// TwinCAT 3 PLC project Untitled1
// ProgramVersion: 3.1.4026.24
// libraries:
//   Tc2_MC2, * (Beckhoff Automation GmbH)
//   Tc2_Standard, * (Beckhoff Automation GmbH)
//   Tc2_System, * (Beckhoff Automation GmbH)
// project tree:
//   DUTs/ ST_ServiceCtrlBase.TcDUT, ST_ServiceStatusBase.TcDUT
//   GVLs/ GVL_Remote.TcGVL
//   / PlcTask.TcTTO
//   POUs/00_BaseUnit/ FB_AxisControl.TcPOU, FB_BaseUnit.TcPOU, T_ResourceOwnerId.TcDUT
//   POUs/10_Module/11_GC/DUTs/ E_GCResourceOwnerId.TcDUT, ST_GC_Admin.TcDUT, ST_GC_ServiceCtrl.TcDUT, ST_GC_ServiceStatus.TcDUT
//   POUs/10_Module/11_GC/DUTs/SpinAxisJogService/ E_GCSpinAxisJogErrorCode.TcDUT, ST_GCSpinAxisJogCtrl.TcDUT, ST_GCSpinAxisJogParam.TcDUT, ST_GCSpinAxisJogStatus.TcDUT
//   POUs/10_Module/11_GC/DUTs/SpinAxisMoveAbsService/ E_GCSpinAxisMoveAbsErrorCode.TcDUT, ST_GCSpinAxisMoveAbsCtrl.TcDUT, ST_GCSpinAxisMoveAbsParam.TcDUT (not stored), ST_GCSpinAxisMoveAbsStatus.TcDUT
//   POUs/10_Module/11_GC/DUTs/SpinAxisMoveVelService/ E_GCSpinAxisMoveVelErrorCode.TcDUT, ST_GCSpinAxisMoveVelCtrl.TcDUT (not stored), ST_GCSpinAxisMoveVelParam.TcDUT, ST_GCSpinAxisMoveVelStatus.TcDUT
//   POUs/10_Module/11_GC/ FB_GC.TcPOU
//   POUs/10_Module/11_GC/Services/ FB_GCSpinAxisJogServices.TcPOU, FB_GCSpinAxisMoveAbsServices.TcPOU, FB_GCSpinAxisMoveVelServices.TcPOU
//   POUs/20_Machine/DUTs/ ST_Machine_Admin.TcDUT, ST_Machine_Ctrl.TcDUT, ST_Machine_ServiceCtrl.TcDUT, ST_Machine_ServiceStatus.TcDUT, ST_Machine_Status.TcDUT
//   POUs/20_Machine/ FB_Machine.TcPOU
//   POUs/ MAIN.TcPOU
//   POUs/PackML_Base/DUTs/ E_PackMLCommand.TcDUT (not stored), E_PackMLHookResult.TcDUT (not stored), E_PackMLMode.TcDUT (not stored), E_PackMLState.TcDUT (not stored), ST_PML_Base_In.TcDUT, ST_PML_Base_Out.TcDUT, T_PackMLMode.TcDUT (not stored)
//   POUs/PackML_Base/ FB_PackMLBase.TcPOU, FB_PackMLModeSet.TcPOU, I_ModuleServiceProperty.TcIO
//   POUs/PackML_Base/Utilities/ F_PackMLCommandToString.TcPOU, F_PackMLModeToString.TcPOU, F_PackMLStateToString.TcPOU (not stored)
// real-time tasks:
//   TASK PlcTask: cycle T#10ms, priority 20, ADS port 350
// motion (NC):
//   TASK NC-Task 1 SAF: cycle T#2ms, priority 4, ADS port 501
//   TASK NC-Task 1 SVB: cycle T#10ms, priority 8, ADS port 511
//   AXIS Axis 1 (id 1)
//     OtherSettings: AllowMotionCmdToSlave=true
//     encoder EncType=1
//     drive DrvType=5
//       Analog: TorqueSetpointScale=10, ScaleFactorActTorque=0.1
//       TimeComp: TaskDelayCycles=1
//     controller CtrType=1
//       CtrPara: PriorControlFactor=1
//         Observer: BandWidth=20
// variable links:
//   Untitled1/Untitled1 Instance <-> NC-Task 1 SAF/Axes/Axis 1
//     PlcTask Inputs/MAIN.Machine._GCSpinAxis.NcToPlc <-> Outputs/ToPlc
//     PlcTask Outputs/MAIN.Machine._GCSpinAxis.PlcToNc <-> Inputs/FromPlc

CONFIGURATION Untitled1
    RESOURCE PLC ON TwinCAT3
        TASK PlcTask(INTERVAL := T#10ms, PRIORITY := 20);
        PROGRAM MAIN WITH PlcTask : MAIN;
    END_RESOURCE
END_CONFIGURATION

// ---- DUTs/ST_ServiceCtrlBase.TcDUT
TYPE ST_ServiceCtrlBase :
STRUCT
	Start : BOOL;
	Reset : BOOL;
	Stop : BOOL;
	Abort : BOOL;
END_STRUCT
END_TYPE

// ---- DUTs/ST_ServiceStatusBase.TcDUT
TYPE ST_ServiceStatusBase :
STRUCT
	Busy : BOOL;
	Done : BOOL;
	Error : BOOL;
	Aborted : BOOL;
	ErrorId : UDINT;
	State : E_PackMLState;
END_STRUCT
END_TYPE

// ---- POUs/00_BaseUnit/T_ResourceOwnerId.TcDUT
// Zero is reserved to represent an unowned resource.
TYPE T_ResourceOwnerId : UDINT;
END_TYPE

// ---- POUs/10_Module/11_GC/DUTs/E_GCResourceOwnerId.TcDUT
{attribute 'qualified_only'}
{attribute 'to_string'}
TYPE E_GCResourceOwnerId :
(
	// Each value identifies one Service instance within the GC Module.
	None := 0,
	SpinAxisJog := 1,
	SpinAxisMoveAbs := 2,
	SpinAxisMoveVel := 3
) UDINT;
END_TYPE

// ---- POUs/10_Module/11_GC/DUTs/SpinAxisJogService/E_GCSpinAxisJogErrorCode.TcDUT
{attribute 'qualified_only'}
{attribute 'to_string'}
TYPE E_GCSpinAxisJogErrorCode :
(
	None := 0,
	Axis_Not_Servo_On_During_Starting,
	Axis_Is_Busy_During_Starting,
	Invalid_Param,
	Jog_Error_During_Execute,
	// The BaseUnit was already owned by another Service.
	Resource_Acquire_Failed_During_Starting
)UDINT;
END_TYPE

// ---- POUs/10_Module/11_GC/DUTs/SpinAxisJogService/ST_GCSpinAxisJogCtrl.TcDUT
TYPE ST_GCSpinAxisJogCtrl EXTENDS ST_ServiceCtrlBase:
STRUCT
	Param : ST_GCSpinAxisJogParam;
END_STRUCT
END_TYPE

// ---- POUs/10_Module/11_GC/DUTs/SpinAxisJogService/ST_GCSpinAxisJogParam.TcDUT
TYPE ST_GCSpinAxisJogParam :
STRUCT
	JogForward : BOOL;
	JogBackwards : BOOL;
	Mode : E_JogMode;
	Position : LREAL;
	Velocity : LREAL;
	Acceleration : LREAL;
	Deceleration : LREAL;
END_STRUCT
END_TYPE

// ---- POUs/10_Module/11_GC/DUTs/SpinAxisJogService/ST_GCSpinAxisJogStatus.TcDUT
TYPE ST_GCSpinAxisJogStatus EXTENDS ST_ServiceStatusBase :
STRUCT
END_STRUCT
END_TYPE

// ---- POUs/10_Module/11_GC/DUTs/SpinAxisMoveAbsService/E_GCSpinAxisMoveAbsErrorCode.TcDUT
{attribute 'qualified_only'}
{attribute 'to_string'}
TYPE E_GCSpinAxisMoveAbsErrorCode :
(
	None := 0,
	Axis_Not_Servo_On_During_Starting,
	Axis_Is_Busy_During_Starting,
	Invalid_Param,
	MoveAbs_Error_During_Execute,
	Error_While_Stop_Axis,
	// The BaseUnit was already owned by another Service.
	Resource_Acquire_Failed_During_Starting
)UDINT;
END_TYPE

// ---- POUs/10_Module/11_GC/DUTs/SpinAxisMoveAbsService/ST_GCSpinAxisMoveAbsCtrl.TcDUT
TYPE ST_GCSpinAxisMoveAbsCtrl EXTENDS ST_ServiceCtrlBase:
STRUCT
	Param : ST_GCSpinAxisMoveAbsParam;
END_STRUCT
END_TYPE

// ---- POUs/10_Module/11_GC/DUTs/SpinAxisMoveAbsService/ST_GCSpinAxisMoveAbsStatus.TcDUT
TYPE ST_GCSpinAxisMoveAbsStatus EXTENDS ST_ServiceStatusBase :
STRUCT
END_STRUCT
END_TYPE

// ---- POUs/10_Module/11_GC/DUTs/SpinAxisMoveVelService/E_GCSpinAxisMoveVelErrorCode.TcDUT
{attribute 'qualified_only'}
{attribute 'to_string'}
TYPE E_GCSpinAxisMoveVelErrorCode :
(
	None := 0,
	Axis_Not_Servo_On_During_Starting,
	Axis_Is_Busy_During_Starting,
	Invalid_Param,
	MoveVel_Error_During_Execute,
	Error_While_Stop_Axis,
	// The BaseUnit was already owned by another Service.
	Resource_Acquire_Failed_During_Starting
)UDINT;
END_TYPE

// ---- POUs/10_Module/11_GC/DUTs/SpinAxisMoveVelService/ST_GCSpinAxisMoveVelParam.TcDUT
TYPE ST_GCSpinAxisMoveVelParam :
STRUCT
	IsPositiveDirection	: BOOL;
	Velocity : LREAL;
	Acceleration : LREAL;
	Deceleration : LREAL;
END_STRUCT
END_TYPE

// ---- POUs/10_Module/11_GC/DUTs/SpinAxisMoveVelService/ST_GCSpinAxisMoveVelStatus.TcDUT
TYPE ST_GCSpinAxisMoveVelStatus EXTENDS ST_ServiceStatusBase :
STRUCT
	ActVel	: LREAL;
END_STRUCT
END_TYPE

// ---- POUs/10_Module/11_GC/DUTs/ST_GC_Admin.TcDUT
TYPE ST_GC_Admin :
STRUCT
	bLocalControl : BOOL;
END_STRUCT
END_TYPE

// ---- POUs/10_Module/11_GC/DUTs/ST_GC_ServiceCtrl.TcDUT
TYPE ST_GC_ServiceCtrl :
STRUCT
	SpinAxisJog : ST_GCSpinAxisJogCtrl;
	SpinAxisMoveAbs : ST_GCSpinAxisMoveAbsCtrl;
	SpinAxisMoveVel	: ST_GCSpinAxisMoveVelCtrl;
END_STRUCT
END_TYPE

// ---- POUs/10_Module/11_GC/DUTs/ST_GC_ServiceStatus.TcDUT
TYPE ST_GC_ServiceStatus :
STRUCT
	SpinAxisJog : ST_GCSpinAxisJogStatus;
	SpinAxisMoveAbs : ST_GCSpinAxisMoveAbsStatus;
	SpinAxisMoveVel : ST_GCSpinAxisMoveVelStatus;
END_STRUCT
END_TYPE

// ---- POUs/20_Machine/DUTs/ST_Machine_Admin.TcDUT
TYPE ST_Machine_Admin :
STRUCT
	GC_Admin : ST_GC_Admin;
END_STRUCT
END_TYPE

// ---- POUs/20_Machine/DUTs/ST_Machine_Ctrl.TcDUT
TYPE ST_Machine_Ctrl:
STRUCT
	Machine_Ctrl :ST_PML_Base_In;
	GC_Ctrl : ST_PML_Base_In;
END_STRUCT
END_TYPE

// ---- POUs/20_Machine/DUTs/ST_Machine_ServiceCtrl.TcDUT
TYPE ST_Machine_ServiceCtrl :
STRUCT
	GC : ST_GC_ServiceCtrl;
END_STRUCT
END_TYPE

// ---- POUs/20_Machine/DUTs/ST_Machine_ServiceStatus.TcDUT
TYPE ST_Machine_ServiceStatus :
STRUCT
	GC : ST_GC_ServiceStatus;
END_STRUCT
END_TYPE

// ---- POUs/20_Machine/DUTs/ST_Machine_Status.TcDUT
TYPE ST_Machine_Status:
STRUCT
	Machine_Status : ST_PML_Base_Out;
	GC_Status : ST_PML_Base_Out;
END_STRUCT
END_TYPE

// ---- POUs/PackML_Base/DUTs/ST_PML_Base_In.TcDUT
TYPE ST_PML_Base_In :
STRUCT
	eCommand				: E_PackMLCommand := E_PackMLCommand.None;
	bCommandChangeRequest	: BOOL;
	eMode					: T_PackMLMode := GVL_PackMLMode.Unknown;
	bModeChangeRequest	: BOOL;
END_STRUCT
END_TYPE

// ---- POUs/PackML_Base/DUTs/ST_PML_Base_Out.TcDUT
TYPE ST_PML_Base_Out :
STRUCT
	eStateCurrent		: E_PackMLState := E_PackMLState.Undefined;
	eStatePrevious		: E_PackMLState := E_PackMLState.Undefined;
	eModeCurrent		: T_PackMLMode := E_PackMLMode.Unknown;
	eModePrevious		: T_PackMLMode := E_PackMLMode.Unknown;

	bCommandAccepted	: BOOL;
	bCommandRejected	: BOOL;

	bModeChanged		: BOOL;
	bModeChangeRejected	: BOOL;
END_STRUCT
END_TYPE

// ---- GVLs/GVL_Remote.TcGVL
{attribute 'qualified_only'}
VAR_GLOBAL
	Ctrl : ST_Machine_Ctrl;
	Status : ST_Machine_Status;
	ServiceCtrl : ST_Machine_ServiceCtrl;
	ServiceStatus : ST_Machine_ServiceStatus;
	Admin : ST_Machine_Admin;
END_VAR

// ---- POUs/PackML_Base/I_ModuleServiceProperty.TcIO
INTERFACE I_ModuleServiceProperty

PROPERTY ModuleMode : T_PackMLMode
GET
END_GET
SET
END_SET
END_PROPERTY

END_INTERFACE

// ---- POUs/MAIN.TcPOU
PROGRAM MAIN
VAR
	Machine : FB_Machine;
END_VAR

Machine(
	Ctrl:= GVL_Remote.Ctrl, 
	Status:= GVL_Remote.Status, 
	ServiceCtrl:= GVL_Remote.ServiceCtrl,
	ServiceStatus:= GVL_Remote.ServiceStatus,
	Admin:= GVL_Remote.Admin);

END_PROGRAM

// ---- POUs/20_Machine/FB_Machine.TcPOU
FUNCTION_BLOCK FB_Machine EXTENDS FB_PackMLModeSet
VAR_INPUT
	Ctrl : REFERENCE TO ST_Machine_Ctrl;
	Status : REFERENCE TO ST_Machine_Status;
	ServiceCtrl : REFERENCE TO ST_Machine_ServiceCtrl;
	ServiceStatus : REFERENCE TO ST_Machine_ServiceStatus;
	Admin : REFERENCE TO ST_Machine_Admin;
END_VAR
VAR_OUTPUT
END_VAR
VAR
	// 有需要特殊操作的需求，所以建立一個ST_Machine_Ctrl變數，讓程式內部可以過一手處理
	_Ctrl : ST_Machine_Ctrl;
	
	// Module
	_GC_Module : FB_GC;
	
	// Component
	_GCSpinAxis : AXIS_REF;
	_GCSpinAxis_BaseUnit : FB_AxisControl;
END_VAR

stIn := Ctrl.Machine_Ctrl;
Status.Machine_Status := stOut;

// Select control source
IF Admin.GC_Admin.bLocalControl THEN
	_Ctrl.GC_Ctrl := Ctrl.GC_Ctrl;
ELSE
	_Ctrl.GC_Ctrl := Ctrl.Machine_Ctrl;
END_IF

A00_BaseUnit();
A01_Module();
A02_CompoundService();

SUPER^();

ACTION A00_BaseUnit:
_GCSpinAxis_BaseUnit(Axis:= _GCSpinAxis);
END_ACTION

ACTION A01_Module:
_GC_Module(
	stIn:= _Ctrl.GC_Ctrl,
	stOut=> Status.GC_Status,
	ServiceCtrl:= ServiceCtrl.GC,
	ServiceStatus:= ServiceStatus.GC,
	Admin:= Admin.GC_Admin,
	SpinAxis_BaseUnit:= _GCSpinAxis_BaseUnit);
END_ACTION

ACTION A02_CompoundService:

END_ACTION

METHOD PROTECTED H_OnAborted
VAR_INPUT
	bFirstScan	: BOOL;
END_VAR
END_METHOD

METHOD PROTECTED H_OnAborting : E_PackMLHookResult
VAR_INPUT
	bFirstScan	: BOOL;
END_VAR
// Default transient hooks complete immediately; override when work is required.
H_OnAborting := E_PackMLHookResult.Done;
END_METHOD

METHOD PROTECTED H_OnClearing : E_PackMLHookResult
VAR_INPUT
	bFirstScan	: BOOL;
END_VAR
H_OnClearing := E_PackMLHookResult.Busy;

// Wait cmd finished
IF Status.GC_Status.eStateCurrent <> E_PackMLState.Stopped THEN
	RETURN;
END_IF

H_OnClearing := E_PackMLHookResult.Done;
END_METHOD

METHOD PROTECTED H_OnComplete
VAR_INPUT
	bFirstScan	: BOOL;
END_VAR
// Default action hook intentionally empty. Override in derived FBs when needed.
END_METHOD

METHOD PROTECTED H_OnCompleting : E_PackMLHookResult
VAR_INPUT
	bFirstScan	: BOOL;
END_VAR
// Default transient hooks complete immediately; override when work is required.
H_OnCompleting := E_PackMLHookResult.Done;
END_METHOD

METHOD PROTECTED H_OnExecute : E_PackMLHookResult
VAR_INPUT
	bFirstScan	: BOOL;
END_VAR
// Execute is stable by default; derived FBs decide when the process is done.
H_OnExecute := E_PackMLHookResult.Busy;
END_METHOD

METHOD PROTECTED H_OnHeld
VAR_INPUT
	bFirstScan	: BOOL;
END_VAR
// Default action hook intentionally empty. Override in derived FBs when needed.
END_METHOD

METHOD PROTECTED H_OnHolding : E_PackMLHookResult
VAR_INPUT
	bFirstScan	: BOOL;
END_VAR
// Default transient hooks complete immediately; override when work is required.
H_OnHolding := E_PackMLHookResult.Done;
END_METHOD

METHOD PROTECTED H_OnIdle
VAR_INPUT
	bFirstScan	: BOOL;
END_VAR
END_METHOD

METHOD PROTECTED H_OnResetting : E_PackMLHookResult
VAR_INPUT
	bFirstScan	: BOOL;
END_VAR
H_OnResetting := E_PackMLHookResult.Busy;

// Wait cmd finished
IF Status.GC_Status.eStateCurrent <> E_PackMLState.Idle THEN
	RETURN;
END_IF

H_OnResetting := E_PackMLHookResult.Done;
END_METHOD

METHOD PROTECTED H_OnStarting : E_PackMLHookResult
VAR_INPUT
	bFirstScan	: BOOL;
END_VAR
H_OnStarting := E_PackMLHookResult.Busy;

// Wait cmd finished
IF Status.GC_Status.eStateCurrent <> E_PackMLState.Execute THEN
	RETURN;
END_IF

H_OnStarting := E_PackMLHookResult.Done;
END_METHOD

METHOD PROTECTED H_OnStopped
VAR_INPUT
	bFirstScan	: BOOL;
END_VAR
END_METHOD

METHOD PROTECTED H_OnStopping : E_PackMLHookResult
VAR_INPUT
	bFirstScan	: BOOL;
END_VAR
H_OnStopping := E_PackMLHookResult.Busy;

// Wait cmd finished
IF Status.GC_Status.eStateCurrent <> E_PackMLState.Stopped THEN
	RETURN;
END_IF

H_OnStopping := E_PackMLHookResult.Done;
END_METHOD

METHOD PROTECTED H_OnSuspended
VAR_INPUT
	bFirstScan	: BOOL;
END_VAR
// Default action hook intentionally empty. Override in derived FBs when needed.
END_METHOD

METHOD PROTECTED H_OnSuspending : E_PackMLHookResult
VAR_INPUT
	bFirstScan	: BOOL;
END_VAR
// Default transient hooks complete immediately; override when work is required.
H_OnSuspending := E_PackMLHookResult.Done;
END_METHOD

METHOD PROTECTED H_OnUndefined : E_PackMLHookResult
VAR_INPUT
	bFirstScan	: BOOL;
END_VAR
// The base FB leaves Undefined immediately unless a derived FB delays startup.
H_OnUndefined := E_PackMLHookResult.Done;
END_METHOD

METHOD PROTECTED H_OnUnholding : E_PackMLHookResult
VAR_INPUT
	bFirstScan	: BOOL;
END_VAR
// Default transient hooks complete immediately; override when work is required.
H_OnUnholding := E_PackMLHookResult.Done;
END_METHOD

METHOD PROTECTED H_OnUnsuspending : E_PackMLHookResult
VAR_INPUT
	bFirstScan	: BOOL;
END_VAR
// Default transient hooks complete immediately; override when work is required.
H_OnUnsuspending := E_PackMLHookResult.Done;
END_METHOD

END_FUNCTION_BLOCK

// ---- POUs/PackML_Base/FB_PackMLModeSet.TcPOU
FUNCTION_BLOCK FB_PackMLModeSet EXTENDS FB_PackMLBase
VAR_INPUT
END_VAR
VAR_OUTPUT
END_VAR
VAR
END_VAR

SUPER^();

METHOD PROTECTED H_IsCommandAllowedByMode : BOOL
VAR_INPUT
	eRequestedCommand	: E_PackMLCommand;
	eActiveMode	: T_PackMLMode;
END_VAR
CASE eActiveMode OF
	GVL_PackMLMode.Manual:
		// Supported commands in manual mode
		CASE eRequestedCommand OF
			E_PackMLCommand.Reset,
			E_PackMLCommand.Start,
			E_PackMLCommand.Stop,
			E_PackMLCommand.Abort,
			E_PackMLCommand.Clear:
				H_IsCommandAllowedByMode := TRUE;
			ELSE
				H_IsCommandAllowedByMode := FALSE;
		END_CASE
	
	GVL_PackMLMode.Production,
	GVL_PackMLMode.Unknown:
		// Support all commands in production mode
		H_IsCommandAllowedByMode := TRUE;
END_CASE
END_METHOD

METHOD PROTECTED H_IsModeSupported : BOOL
VAR_INPUT
	eRequestedMode	: T_PackMLMode;
END_VAR
CASE eRequestedMode OF
	GVL_PackMLMode.Manual,
	GVL_PackMLMode.Production:
		H_IsModeSupported := TRUE;

	ELSE
		H_IsModeSupported := FALSE;
END_CASE
END_METHOD

METHOD PROTECTED H_IsStateSupportedByMode : BOOL
VAR_INPUT
	eRequestedMode	: T_PackMLMode;
	eCurrentState	: E_PackMLState;
END_VAR
CASE eRequestedMode OF
	
	GVL_PackMLMode.Manual:
		// Support states in manual mode
		CASE eCurrentState OF
			E_PackMLState.Idle,
			E_PackMLState.Starting,
			E_PackMLState.Execute,
			E_PackMLState.Aborting,
			E_PackMLState.Aborted,
			E_PackMLState.Clearing,
			E_PackMLState.Stopped,
			E_PackMLState.Resetting:
			H_IsStateSupportedByMode := TRUE;
			
			ELSE
				H_IsStateSupportedByMode := FALSE;
		END_CASE
		
	
	GVL_PackMLMode.Production,
	GVL_PackMLMode.Unknown:
		// Support all state in production mode
		H_IsStateSupportedByMode := TRUE;
END_CASE
END_METHOD

END_FUNCTION_BLOCK

// ---- POUs/PackML_Base/FB_PackMLBase.TcPOU
FUNCTION_BLOCK FB_PackMLBase
VAR_INPUT
	stIn	: ST_PML_Base_In;
	
	bEnable				: BOOL := TRUE;
	bExternalFault		: BOOL;
END_VAR
VAR_OUTPUT
	stOut	: ST_PML_Base_Out;
	
	sStateErrorText		: STRING(255);
	sModeErrorText		: STRING(255);
	bTransitionActive	: BOOL;
END_VAR
VAR
	_eLastCommand			: E_PackMLCommand := E_PackMLCommand.None;
	_eCommandToProcess		: E_PackMLCommand := E_PackMLCommand.None;
	_eQueuedCommand			: E_PackMLCommand := E_PackMLCommand.None;
	_bQueuedCommandRequest	: BOOL;
	_bCommandConsumed		: BOOL;
	_bModeChangeConsumed	: BOOL;
	_bStateFirstScan		: BOOL := TRUE;
	_bStateFirstScanForHook	: BOOL;
	_eHookResult			: E_PackMLHookResult;
END_VAR

// Reset edge-style status before evaluating this PLC cycle.
_eCommandToProcess		:= E_PackMLCommand.None;

// Command and mode request feedback is latched for HMI/upper-layer handshakes
// until the corresponding request input returns to FALSE.
IF NOT stIn.bCommandChangeRequest THEN
	stOut.bCommandAccepted	:= FALSE;
	stOut.bCommandRejected	:= FALSE;
	sStateErrorText			:= '';
END_IF

IF NOT stIn.bModeChangeRequest THEN
	stOut.bModeChanged		:= FALSE;
	stOut.bModeChangeRejected	:= FALSE;
	sModeErrorText		:= '';
END_IF

// A disabled base FB holds the current state and suppresses transition activity.
IF NOT bEnable THEN
	bTransitionActive := FALSE;
	RETURN;
END_IF

// Mode change requests are edge/latch based, matching command request behavior.
// The caller must clear stIn.bModeChangeRequest before the same request can run again.
IF NOT stIn.bModeChangeRequest THEN
	_bModeChangeConsumed := FALSE;
END_IF

IF stIn.bModeChangeRequest AND NOT _bModeChangeConsumed THEN
	_bModeChangeConsumed := TRUE;

	IF NOT H_IsModeSupported(stIn.eMode) THEN
		M_RejectModeChange('Requested mode is not supported.');
	ELSIF stIn.eMode = stOut.eModeCurrent THEN
		M_RejectModeChange('Requested mode is already active.');
	ELSIF NOT M_IsModeChangeAllowedByState() THEN
		M_RejectModeChange('Mode change is only allowed from Aborted, Stopped, Idle, or Complete.');
	ELSIF NOT H_IsStateSupportedByMode(stIn.eMode, stOut.eStateCurrent) THEN
		M_RejectModeChange('Requested mode does not support the current PackML state.');
	ELSE
		M_ChangeMode(stIn.eMode);
	END_IF
END_IF

// Command requests are edge/latch based, matching mode-change request behavior.
// The caller must clear stIn.bCommandChangeRequest before another command can run.
IF NOT stIn.bCommandChangeRequest THEN
	_bCommandConsumed	:= FALSE;
	_eLastCommand		:= E_PackMLCommand.None;
END_IF

// External faults have priority over normal commands and force the abort path
// only while the machine is not already Aborting or Aborted.
IF bExternalFault AND M_IsAbortAllowedByState() THEN
	_eCommandToProcess := E_PackMLCommand.Abort;
ELSIF _bQueuedCommandRequest AND (_eQueuedCommand <> E_PackMLCommand.None) THEN
	_eCommandToProcess		:= _eQueuedCommand;
	_eQueuedCommand			:= E_PackMLCommand.None;
	_bQueuedCommandRequest	:= FALSE;
ELSIF stIn.bCommandChangeRequest AND (stIn.eCommand <> E_PackMLCommand.None) AND NOT _bCommandConsumed THEN
	_eCommandToProcess	:= stIn.eCommand;
	_eLastCommand		:= stIn.eCommand;
	_bCommandConsumed	:= TRUE;
END_IF

// Mode policy hooks run before PackML state guards so a forbidden command reports
// the mode reason instead of a state reason.
IF (_eCommandToProcess <> E_PackMLCommand.None) AND NOT H_IsCommandAllowedByMode(_eCommandToProcess, stOut.eModeCurrent) THEN
	M_RejectCommand(M_BuildCommandRejectedByModeText(_eCommandToProcess, stOut.eModeCurrent));
	_eCommandToProcess := E_PackMLCommand.None;
END_IF

// Dispatch the accepted command through private PackML state guards.
// Rejected commands never mutate the state and return a readable error text.
CASE _eCommandToProcess OF
	E_PackMLCommand.Clear:
		IF M_IsClearAllowedByState() THEN
			stOut.bCommandAccepted := TRUE;
			M_ChangeState(E_PackMLState.Clearing);
		ELSE
			M_RejectCommand('Clear command is only valid from Aborted.');
		END_IF

	E_PackMLCommand.Reset:
		IF M_IsResetAllowedByState() THEN
			stOut.bCommandAccepted := TRUE;
			M_ChangeState(E_PackMLState.Resetting);
		ELSE
			M_RejectCommand('Reset command is only valid from Stopped or Complete.');
		END_IF

	E_PackMLCommand.Start:
		IF M_IsStartAllowedByState() THEN
			stOut.bCommandAccepted := TRUE;
			M_ChangeState(E_PackMLState.Starting);
		ELSE
			M_RejectCommand('Start command is only valid from Idle.');
		END_IF

	E_PackMLCommand.Stop:
		IF M_IsStopAllowedByState() THEN
			stOut.bCommandAccepted := TRUE;
			M_ChangeState(E_PackMLState.Stopping);
		ELSE
			M_RejectCommand('Stop command is not valid from the current PackML state.');
		END_IF

	E_PackMLCommand.Hold:
		IF M_IsHoldAllowedByState() THEN
			stOut.bCommandAccepted := TRUE;
			M_ChangeState(E_PackMLState.Holding);
		ELSE
			M_RejectCommand('Hold command is only valid from Execute.');
		END_IF

	E_PackMLCommand.Unhold:
		IF M_IsUnholdAllowedByState() THEN
			stOut.bCommandAccepted := TRUE;
			M_ChangeState(E_PackMLState.Unholding);
		ELSE
			M_RejectCommand('Unhold command is only valid from Held.');
		END_IF

	E_PackMLCommand.Suspend:
		IF M_IsSuspendAllowedByState() THEN
			stOut.bCommandAccepted := TRUE;
			M_ChangeState(E_PackMLState.Suspending);
		ELSE
			M_RejectCommand('Suspend command is only valid from Execute.');
		END_IF

	E_PackMLCommand.Unsuspend:
		IF M_IsUnsuspendAllowedByState() THEN
			stOut.bCommandAccepted := TRUE;
			M_ChangeState(E_PackMLState.Unsuspending);
		ELSE
			M_RejectCommand('Unsuspend command is only valid from Suspended.');
		END_IF

	E_PackMLCommand.Abort:
		IF M_IsAbortAllowedByState() THEN
			stOut.bCommandAccepted := TRUE;
			M_ChangeState(E_PackMLState.Aborting);
		ELSE
			M_RejectCommand('Abort command is not valid while already Aborting or Aborted.');
		END_IF
END_CASE

// Run the current state's action hook, then advance transient states when their
// hook reports Done. Stable states remain active until a command moves them.
_bStateFirstScanForHook	:= _bStateFirstScan;
_bStateFirstScan		:= FALSE;

CASE stOut.eStateCurrent OF
	E_PackMLState.Undefined:
		_eHookResult := H_OnUndefined(_bStateFirstScanForHook);
		IF _eHookResult = E_PackMLHookResult.Done THEN
			M_ChangeState(E_PackMLState.Aborted);
		END_IF

	E_PackMLState.Clearing:
		_eHookResult := H_OnClearing(_bStateFirstScanForHook);
		IF _eHookResult = E_PackMLHookResult.Done THEN
			M_ChangeState(E_PackMLState.Stopped);
		END_IF

	E_PackMLState.Stopped:
		H_OnStopped(_bStateFirstScanForHook);

	E_PackMLState.Starting:
		_eHookResult := H_OnStarting(_bStateFirstScanForHook);
		IF _eHookResult = E_PackMLHookResult.Done THEN
			M_ChangeState(E_PackMLState.Execute);
		END_IF

	E_PackMLState.Idle:
		H_OnIdle(_bStateFirstScanForHook);

	E_PackMLState.Suspended:
		H_OnSuspended(_bStateFirstScanForHook);

	E_PackMLState.Execute:
		_eHookResult := H_OnExecute(_bStateFirstScanForHook);
		IF _eHookResult = E_PackMLHookResult.Done THEN
			M_ChangeState(E_PackMLState.Completing);
		END_IF

	E_PackMLState.Stopping:
		_eHookResult := H_OnStopping(_bStateFirstScanForHook);
		IF _eHookResult = E_PackMLHookResult.Done THEN
			M_ChangeState(E_PackMLState.Stopped);
		END_IF

	E_PackMLState.Aborting:
		_eHookResult := H_OnAborting(_bStateFirstScanForHook);
		IF _eHookResult = E_PackMLHookResult.Done THEN
			M_ChangeState(E_PackMLState.Aborted);
		END_IF

	E_PackMLState.Aborted:
		H_OnAborted(_bStateFirstScanForHook);

	E_PackMLState.Holding:
		_eHookResult := H_OnHolding(_bStateFirstScanForHook);
		IF _eHookResult = E_PackMLHookResult.Done THEN
			M_ChangeState(E_PackMLState.Held);
		END_IF

	E_PackMLState.Held:
		H_OnHeld(_bStateFirstScanForHook);

	E_PackMLState.Unholding:
		_eHookResult := H_OnUnholding(_bStateFirstScanForHook);
		IF _eHookResult = E_PackMLHookResult.Done THEN
			M_ChangeState(E_PackMLState.Execute);
		END_IF

	E_PackMLState.Suspending:
		_eHookResult := H_OnSuspending(_bStateFirstScanForHook);
		IF _eHookResult = E_PackMLHookResult.Done THEN
			M_ChangeState(E_PackMLState.Suspended);
		END_IF

	E_PackMLState.Unsuspending:
		_eHookResult := H_OnUnsuspending(_bStateFirstScanForHook);
		IF _eHookResult = E_PackMLHookResult.Done THEN
			M_ChangeState(E_PackMLState.Execute);
		END_IF

	E_PackMLState.Resetting:
		_eHookResult := H_OnResetting(_bStateFirstScanForHook);
		IF _eHookResult = E_PackMLHookResult.Done THEN
			M_ChangeState(E_PackMLState.Idle);
		END_IF

	E_PackMLState.Completing:
		_eHookResult := H_OnCompleting(_bStateFirstScanForHook);
		IF _eHookResult = E_PackMLHookResult.Done THEN
			M_ChangeState(E_PackMLState.Complete);
		END_IF

	E_PackMLState.Complete:
		H_OnComplete(_bStateFirstScanForHook);
END_CASE

// Transition activity is true for transient states that normally need completion
// confirmation from their state hook.
bTransitionActive :=
	(stOut.eStateCurrent = E_PackMLState.Undefined) OR
	(stOut.eStateCurrent = E_PackMLState.Clearing) OR
	(stOut.eStateCurrent = E_PackMLState.Starting) OR
	(stOut.eStateCurrent = E_PackMLState.Stopping) OR
	(stOut.eStateCurrent = E_PackMLState.Aborting) OR
	(stOut.eStateCurrent = E_PackMLState.Holding) OR
	(stOut.eStateCurrent = E_PackMLState.Unholding) OR
	(stOut.eStateCurrent = E_PackMLState.Suspending) OR
	(stOut.eStateCurrent = E_PackMLState.Unsuspending) OR
	(stOut.eStateCurrent = E_PackMLState.Resetting) OR
	(stOut.eStateCurrent = E_PackMLState.Completing);

METHOD PROTECTED H_IsCommandAllowedByMode : BOOL
VAR_INPUT
	eRequestedCommand	: E_PackMLCommand;
	eActiveMode			: T_PackMLMode;
END_VAR
// Modes are application-defined in library use; override to restrict commands per mode.
H_IsCommandAllowedByMode := TRUE;
END_METHOD

METHOD PROTECTED H_IsModeSupported : BOOL
VAR_INPUT
	eRequestedMode	: T_PackMLMode;
END_VAR
// Modes are application-defined in library use; override to reject unsupported modes.
H_IsModeSupported := TRUE;
END_METHOD

METHOD PROTECTED H_IsStateSupportedByMode : BOOL
VAR_INPUT
	eRequestedMode	: T_PackMLMode;
	eCurrentState	: E_PackMLState;
END_VAR
// Modes are application-defined in library use; override to restrict mode/state pairs.
H_IsStateSupportedByMode := TRUE;
END_METHOD

METHOD PROTECTED H_OnAborted
VAR_INPUT
	bFirstScan	: BOOL;
END_VAR
// Default action hook intentionally empty. Override in derived FBs when needed.
END_METHOD

METHOD PROTECTED H_OnAborting : E_PackMLHookResult
VAR_INPUT
	bFirstScan	: BOOL;
END_VAR
// Default transient hooks complete immediately; override when work is required.
H_OnAborting := E_PackMLHookResult.Done;
END_METHOD

METHOD PROTECTED H_OnClearing : E_PackMLHookResult
VAR_INPUT
	bFirstScan	: BOOL;
END_VAR
// Default transient hooks complete immediately; override when work is required.
H_OnClearing := E_PackMLHookResult.Done;
END_METHOD

METHOD PROTECTED H_OnComplete
VAR_INPUT
	bFirstScan	: BOOL;
END_VAR
// Default action hook intentionally empty. Override in derived FBs when needed.
END_METHOD

METHOD PROTECTED H_OnCompleting : E_PackMLHookResult
VAR_INPUT
	bFirstScan	: BOOL;
END_VAR
// Default transient hooks complete immediately; override when work is required.
H_OnCompleting := E_PackMLHookResult.Done;
END_METHOD

METHOD PROTECTED H_OnExecute : E_PackMLHookResult
VAR_INPUT
	bFirstScan	: BOOL;
END_VAR
// Execute is stable by default; derived FBs decide when the process is done.
H_OnExecute := E_PackMLHookResult.Busy;
END_METHOD

METHOD PROTECTED H_OnHeld
VAR_INPUT
	bFirstScan	: BOOL;
END_VAR
// Default action hook intentionally empty. Override in derived FBs when needed.
END_METHOD

METHOD PROTECTED H_OnHolding : E_PackMLHookResult
VAR_INPUT
	bFirstScan	: BOOL;
END_VAR
// Default transient hooks complete immediately; override when work is required.
H_OnHolding := E_PackMLHookResult.Done;
END_METHOD

METHOD PROTECTED H_OnIdle
VAR_INPUT
	bFirstScan	: BOOL;
END_VAR
// Default action hook intentionally empty. Override in derived FBs when needed.
END_METHOD

METHOD PROTECTED H_OnModeChanged
VAR_INPUT
	ePreviousMode	: T_PackMLMode;
	eNewMode		: T_PackMLMode;
END_VAR
// Default mode-change hook intentionally empty. Override in derived FBs when needed.
END_METHOD

METHOD PROTECTED H_OnResetting : E_PackMLHookResult
VAR_INPUT
	bFirstScan	: BOOL;
END_VAR
// Default transient hooks complete immediately; override when work is required.
H_OnResetting := E_PackMLHookResult.Done;
END_METHOD

METHOD PROTECTED H_OnStarting : E_PackMLHookResult
VAR_INPUT
	bFirstScan	: BOOL;
END_VAR
// Default transient hooks complete immediately; override when work is required.
H_OnStarting := E_PackMLHookResult.Done;
END_METHOD

METHOD PROTECTED H_OnStateChanged
VAR_INPUT
	ePreviousState	: E_PackMLState;
	eNewState		: E_PackMLState;
END_VAR
// Default state-change hook intentionally empty. Override in derived FBs when needed.
END_METHOD

METHOD PROTECTED H_OnStopped
VAR_INPUT
	bFirstScan	: BOOL;
END_VAR
// Default action hook intentionally empty. Override in derived FBs when needed.
END_METHOD

METHOD PROTECTED H_OnStopping : E_PackMLHookResult
VAR_INPUT
	bFirstScan	: BOOL;
END_VAR
// Default transient hooks complete immediately; override when work is required.
H_OnStopping := E_PackMLHookResult.Done;
END_METHOD

METHOD PROTECTED H_OnSuspended
VAR_INPUT
	bFirstScan	: BOOL;
END_VAR
// Default action hook intentionally empty. Override in derived FBs when needed.
END_METHOD

METHOD PROTECTED H_OnSuspending : E_PackMLHookResult
VAR_INPUT
	bFirstScan	: BOOL;
END_VAR
// Default transient hooks complete immediately; override when work is required.
H_OnSuspending := E_PackMLHookResult.Done;
END_METHOD

METHOD PROTECTED H_OnUndefined : E_PackMLHookResult
VAR_INPUT
	bFirstScan	: BOOL;
END_VAR
// The base FB leaves Undefined immediately unless a derived FB delays startup.
H_OnUndefined := E_PackMLHookResult.Done;
END_METHOD

METHOD PROTECTED H_OnUnholding : E_PackMLHookResult
VAR_INPUT
	bFirstScan	: BOOL;
END_VAR
// Default transient hooks complete immediately; override when work is required.
H_OnUnholding := E_PackMLHookResult.Done;
END_METHOD

METHOD PROTECTED H_OnUnsuspending : E_PackMLHookResult
VAR_INPUT
	bFirstScan	: BOOL;
END_VAR
// Default transient hooks complete immediately; override when work is required.
H_OnUnsuspending := E_PackMLHookResult.Done;
END_METHOD

METHOD PRIVATE M_BuildCommandRejectedByModeText : STRING(255)
VAR_INPUT
	eRejectedCommand	: E_PackMLCommand;
	eActiveMode			: T_PackMLMode;
END_VAR
// Build the rejection text from display names so HMI text stays operator-friendly.
M_BuildCommandRejectedByModeText := CONCAT(F_PackMLCommandToString(eRejectedCommand), ' command is not allowed in ');
M_BuildCommandRejectedByModeText := CONCAT(M_BuildCommandRejectedByModeText, F_PackMLModeToString(eActiveMode));
M_BuildCommandRejectedByModeText := CONCAT(M_BuildCommandRejectedByModeText, ' mode.');
END_METHOD

METHOD PRIVATE M_ChangeMode
VAR_INPUT
	eNextMode	: T_PackMLMode;
END_VAR
// Centralize mode mutation so previous-mode and edge outputs stay consistent.
IF stOut.eModeCurrent <> eNextMode THEN
	stOut.eModePrevious	:= stOut.eModeCurrent;
	stOut.eModeCurrent	:= eNextMode;
	stOut.bModeChanged	:= TRUE;
	H_OnModeChanged(stOut.eModePrevious, stOut.eModeCurrent);
END_IF
END_METHOD

METHOD PRIVATE M_ChangeState
VAR_INPUT
	eNextState	: E_PackMLState;
END_VAR
// Centralize state mutation so previous-state and edge outputs stay consistent.
IF stOut.eStateCurrent <> eNextState THEN
	stOut.eStatePrevious	:= stOut.eStateCurrent;
	stOut.eStateCurrent			:= eNextState;
	_bStateFirstScan			:= TRUE;
	H_OnStateChanged(stOut.eStatePrevious, stOut.eStateCurrent);
END_IF
END_METHOD

METHOD PRIVATE M_IsAbortAllowedByState : BOOL
// Abort is valid from every state except the terminal abort states.
M_IsAbortAllowedByState := (stOut.eStateCurrent <> E_PackMLState.Aborting) AND (stOut.eStateCurrent <> E_PackMLState.Aborted);
END_METHOD

METHOD PRIVATE M_IsClearAllowedByState : BOOL
// Clear leaves the safe Aborted state and starts the resettable stop path.
M_IsClearAllowedByState := stOut.eStateCurrent = E_PackMLState.Aborted;
END_METHOD

METHOD PRIVATE M_IsCompleteAllowedByState : BOOL
// Complete is only meaningful while the unit is executing.
M_IsCompleteAllowedByState := stOut.eStateCurrent = E_PackMLState.Execute;
END_METHOD

METHOD PRIVATE M_IsHoldAllowedByState : BOOL
// Hold pauses an active Execute flow.
M_IsHoldAllowedByState := stOut.eStateCurrent = E_PackMLState.Execute;
END_METHOD

METHOD PRIVATE M_IsModeChangeAllowedByState : BOOL
// Mode changes can only be attempted from safe stable states.
// Target mode compatibility is checked separately after this safety gate.
// Henry: Bypass "Held" & "Suspended" state due to consideration about state-related parameters inconsistent
M_IsModeChangeAllowedByState :=
	(stOut.eStateCurrent = E_PackMLState.Aborted) OR
	(stOut.eStateCurrent = E_PackMLState.Stopped) OR
	(stOut.eStateCurrent = E_PackMLState.Idle) OR
	(stOut.eStateCurrent = E_PackMLState.Complete);
END_METHOD

METHOD PRIVATE M_IsResetAllowedByState : BOOL
// Reset prepares the unit from Stopped or Complete into Idle.
M_IsResetAllowedByState := (stOut.eStateCurrent = E_PackMLState.Stopped) OR (stOut.eStateCurrent = E_PackMLState.Complete);
END_METHOD

METHOD PRIVATE M_IsStartAllowedByState : BOOL
// Start begins production or operation only from Idle.
M_IsStartAllowedByState := stOut.eStateCurrent = E_PackMLState.Idle;
END_METHOD

METHOD PRIVATE M_IsStopAllowedByState : BOOL
// Stop is accepted from normal operating, paused, and completing states.
M_IsStopAllowedByState :=
	(stOut.eStateCurrent = E_PackMLState.Starting) OR
	(stOut.eStateCurrent = E_PackMLState.Idle) OR
	(stOut.eStateCurrent = E_PackMLState.Execute) OR
	(stOut.eStateCurrent = E_PackMLState.Completing) OR
	(stOut.eStateCurrent = E_PackMLState.Complete) OR
	(stOut.eStateCurrent = E_PackMLState.Holding) OR
	(stOut.eStateCurrent = E_PackMLState.Held) OR
	(stOut.eStateCurrent = E_PackMLState.Unholding) OR
	(stOut.eStateCurrent = E_PackMLState.Suspending) OR
	(stOut.eStateCurrent = E_PackMLState.Suspended) OR
	(stOut.eStateCurrent = E_PackMLState.Unsuspending);
END_METHOD

METHOD PRIVATE M_IsSuspendAllowedByState : BOOL
// Suspend pauses Execute because of an external process condition.
M_IsSuspendAllowedByState := stOut.eStateCurrent = E_PackMLState.Execute;
END_METHOD

METHOD PRIVATE M_IsUnholdAllowedByState : BOOL
// Unhold resumes from the stable Held state.
M_IsUnholdAllowedByState := stOut.eStateCurrent = E_PackMLState.Held;
END_METHOD

METHOD PRIVATE M_IsUnsuspendAllowedByState : BOOL
// Unsuspend resumes from the stable Suspended state.
M_IsUnsuspendAllowedByState := stOut.eStateCurrent = E_PackMLState.Suspended;
END_METHOD

METHOD PRIVATE M_RejectCommand
VAR_INPUT
	sText	: STRING(255);
END_VAR
// Centralize rejected-command reporting so every guard failure has text.
stOut.bCommandRejected	:= TRUE;
sStateErrorText		:= sText;
END_METHOD

METHOD PRIVATE M_RejectModeChange
VAR_INPUT
	sText	: STRING(255);
END_VAR
// Keep mode-change errors separate from PackML command/state errors.
stOut.bModeChangeRejected	:= TRUE;
sModeErrorText		:= sText;
END_METHOD

// Used for requesting PackML command inside state machine itself 
METHOD PROTECTED RequestCommand : BOOL
VAR_INPUT
	eTargetCmd	: E_PackMLCommand;
END_VAR
RequestCommand := FALSE;

IF _bQueuedCommandRequest OR stIn.bModeChangeRequest THEN
	RETURN;
END_IF

_eQueuedCommand			:= eTargetCmd;
_bQueuedCommandRequest	:= TRUE;
RequestCommand := TRUE;
END_METHOD

END_FUNCTION_BLOCK

// ---- POUs/PackML_Base/Utilities/F_PackMLCommandToString.TcPOU
FUNCTION F_PackMLCommandToString : STRING(80)
VAR_INPUT
	eCommand	: E_PackMLCommand;
END_VAR

CASE eCommand OF
	E_PackMLCommand.None:
		F_PackMLCommandToString := 'None';
	E_PackMLCommand.Reset:
		F_PackMLCommandToString := 'Reset';
	E_PackMLCommand.Start:
		F_PackMLCommandToString := 'Start';
	E_PackMLCommand.Stop:
		F_PackMLCommandToString := 'Stop';
	E_PackMLCommand.Hold:
		F_PackMLCommandToString := 'Hold';
	E_PackMLCommand.Unhold:
		F_PackMLCommandToString := 'Unhold';
	E_PackMLCommand.Suspend:
		F_PackMLCommandToString := 'Suspend';
	E_PackMLCommand.Unsuspend:
		F_PackMLCommandToString := 'Unsuspend';
	E_PackMLCommand.Abort:
		F_PackMLCommandToString := 'Abort';
	E_PackMLCommand.Clear:
		F_PackMLCommandToString := 'Clear';
ELSE
	F_PackMLCommandToString := 'Unknown';
END_CASE

END_FUNCTION

// ---- POUs/PackML_Base/Utilities/F_PackMLModeToString.TcPOU
FUNCTION F_PackMLModeToString : STRING(80)
VAR_INPUT
	eMode	: T_PackMLMode;
END_VAR

CASE eMode OF
	E_PackMLMode.Unknown:
		F_PackMLModeToString := 'Unknown';
	E_PackMLMode.Production:
		F_PackMLModeToString := 'Production';
	E_PackMLMode.Manual:
		F_PackMLModeToString := 'Manual';
ELSE
	F_PackMLModeToString := CONCAT('Mode ', UINT_TO_STRING(eMode));
END_CASE

END_FUNCTION

// ---- POUs/10_Module/11_GC/FB_GC.TcPOU
FUNCTION_BLOCK FB_GC EXTENDS FB_PackMLModeSet
VAR_INPUT
	ServiceCtrl : REFERENCE TO ST_GC_ServiceCtrl;
	ServiceStatus : REFERENCE TO ST_GC_ServiceStatus;
	Admin : REFERENCE TO ST_GC_Admin;
	
	// Base unit used in GC chamber
	SpinAxis_BaseUnit : REFERENCE TO FB_AxisControl;
END_VAR

VAR_OUTPUT
	
END_VAR

VAR
	// 有需要特殊操作的需求，所以建立一個 ST_GC_ServiceCtrl 變數，讓程式內部可以過一手處理
	_ServiceCtrl : ST_GC_ServiceCtrl;
	_SpinAxisJogService : FB_GCSpinAxisJogServices;
	_SpinAxisMoveAbsService : FB_GCSpinAxisMoveAbsServices;
	_SpinAxisMoveVelService : FB_GCSpinAxisMoveVelServices;
END_VAR

A00_Service();
SUPER^();

ACTION A00_Service:
_SpinAxisJogService(
	Ctrl:= _ServiceCtrl.SpinAxisJog,
	Status:= ServiceStatus.SpinAxisJog,
	Axis_BaseUnit:= SpinAxis_BaseUnit,
	// Owner IDs are assigned by the Module so each Service instance is unique.
	ResourceOwnerId:= E_GCResourceOwnerId.SpinAxisJog);

_SpinAxisMoveAbsService(
	Ctrl:= _ServiceCtrl.SpinAxisMoveAbs,
	Status:= ServiceStatus.SpinAxisMoveAbs,
	Axis_BaseUnit:= SpinAxis_BaseUnit,
	ResourceOwnerId:= E_GCResourceOwnerId.SpinAxisMoveAbs);

_SpinAxisMoveVelService(
	Ctrl:= _ServiceCtrl.SpinAxisMoveVel,
	Status:= ServiceStatus.SpinAxisMoveVel,
	Axis_BaseUnit:= SpinAxis_BaseUnit,
	ResourceOwnerId:= E_GCResourceOwnerId.SpinAxisMoveVel);
END_ACTION

METHOD PROTECTED H_OnAborted
VAR_INPUT
	bFirstScan	: BOOL;
END_VAR
// Default action hook intentionally empty. Override in derived FBs when needed.
END_METHOD

METHOD PROTECTED H_OnAborting : E_PackMLHookResult
VAR_INPUT
	bFirstScan	: BOOL;
END_VAR
// Default transient hooks complete immediately; override when work is required.
H_OnAborting := E_PackMLHookResult.Done;
END_METHOD

METHOD PROTECTED H_OnClearing : E_PackMLHookResult
VAR_INPUT
	bFirstScan	: BOOL;
END_VAR
H_OnClearing := E_PackMLHookResult.Done;
END_METHOD

METHOD PROTECTED H_OnComplete
VAR_INPUT
	bFirstScan	: BOOL;
END_VAR
// Default action hook intentionally empty. Override in derived FBs when needed.
END_METHOD

METHOD PROTECTED H_OnCompleting : E_PackMLHookResult
VAR_INPUT
	bFirstScan	: BOOL;
END_VAR
// Default transient hooks complete immediately; override when work is required.
H_OnCompleting := E_PackMLHookResult.Done;
END_METHOD

METHOD PROTECTED H_OnExecute : E_PackMLHookResult
VAR_INPUT
	bFirstScan	: BOOL;
END_VAR
// Execute is stable by default; derived FBs decide when the process is done.
H_OnExecute := E_PackMLHookResult.Busy;

// Mapping control data
_ServiceCtrl := ServiceCtrl;
END_METHOD

METHOD PROTECTED H_OnHeld
VAR_INPUT
	bFirstScan	: BOOL;
END_VAR
// Default action hook intentionally empty. Override in derived FBs when needed.
END_METHOD

METHOD PROTECTED H_OnHolding : E_PackMLHookResult
VAR_INPUT
	bFirstScan	: BOOL;
END_VAR
// Default transient hooks complete immediately; override when work is required.
H_OnHolding := E_PackMLHookResult.Done;
END_METHOD

METHOD PROTECTED H_OnIdle
VAR_INPUT
	bFirstScan	: BOOL;
END_VAR
// Default action hook intentionally empty. Override in derived FBs when needed.
END_METHOD

METHOD PROTECTED H_OnModeChanged
VAR_INPUT
	ePreviousMode	: T_PackMLMode;
	eNewMode	: T_PackMLMode;
END_VAR
// Notice current mode to each service
_SpinAxisJogService.ModuleMode := eNewMode;
_SpinAxisMoveAbsService.ModuleMode := eNewMode;
_SpinAxisMoveVelService.ModuleMode := eNewMode;
END_METHOD

METHOD PROTECTED H_OnResetting : E_PackMLHookResult
VAR_INPUT
	bFirstScan	: BOOL;
END_VAR
H_OnResetting := E_PackMLHookResult.Busy;

// Request reset cmd to services
_ServiceCtrl.SpinAxisJog.Reset := TRUE;
_ServiceCtrl.SpinAxisMoveAbs.Reset := TRUE;
_ServiceCtrl.SpinAxisMoveVel.Reset := TRUE;

// Wait cmd finished
IF ServiceStatus.SpinAxisJog.State <> E_PackMLState.Idle
	OR ServiceStatus.SpinAxisMoveAbs.State <> E_PackMLState.Idle
	OR ServiceStatus.SpinAxisMoveVel.State <> E_PackMLState.Idle THEN
	RETURN;
END_IF

// Reset trigger
_ServiceCtrl.SpinAxisJog.Reset := FALSE;
_ServiceCtrl.SpinAxisMoveAbs.Reset := FALSE;
_ServiceCtrl.SpinAxisMoveVel.Reset := FALSE;

H_OnResetting := E_PackMLHookResult.Done;
END_METHOD

METHOD PROTECTED H_OnStarting : E_PackMLHookResult
VAR_INPUT
	bFirstScan	: BOOL;
END_VAR
// Default transient hooks complete immediately; override when work is required.
H_OnStarting := E_PackMLHookResult.Done;
END_METHOD

METHOD PROTECTED H_OnStopped
VAR_INPUT
	bFirstScan	: BOOL;
END_VAR
// Default action hook intentionally empty. Override in derived FBs when needed.
END_METHOD

METHOD PROTECTED H_OnStopping : E_PackMLHookResult
VAR_INPUT
	bFirstScan	: BOOL;
END_VAR
// Default transient hooks complete immediately; override when work is required.
H_OnStopping := E_PackMLHookResult.Done;
END_METHOD

METHOD PROTECTED H_OnSuspended
VAR_INPUT
	bFirstScan	: BOOL;
END_VAR
// Default action hook intentionally empty. Override in derived FBs when needed.
END_METHOD

METHOD PROTECTED H_OnSuspending : E_PackMLHookResult
VAR_INPUT
	bFirstScan	: BOOL;
END_VAR
// Default transient hooks complete immediately; override when work is required.
H_OnSuspending := E_PackMLHookResult.Done;
END_METHOD

METHOD PROTECTED H_OnUndefined : E_PackMLHookResult
VAR_INPUT
	bFirstScan	: BOOL;
END_VAR
// The base FB leaves Undefined immediately unless a derived FB delays startup.
H_OnUndefined := E_PackMLHookResult.Done;
END_METHOD

METHOD PROTECTED H_OnUnholding : E_PackMLHookResult
VAR_INPUT
	bFirstScan	: BOOL;
END_VAR
// Default transient hooks complete immediately; override when work is required.
H_OnUnholding := E_PackMLHookResult.Done;
END_METHOD

METHOD PROTECTED H_OnUnsuspending : E_PackMLHookResult
VAR_INPUT
	bFirstScan	: BOOL;
END_VAR
// Default transient hooks complete immediately; override when work is required.
H_OnUnsuspending := E_PackMLHookResult.Done;
END_METHOD

END_FUNCTION_BLOCK

// ---- POUs/00_BaseUnit/FB_AxisControl.TcPOU
FUNCTION_BLOCK FB_AxisControl EXTENDS FB_BaseUnit
VAR_INPUT
	Axis	: REFERENCE TO AXIS_REF;
END_VAR

VAR_OUTPUT
	ErrorText : STRING;
END_VAR

VAR
	_MCMoveAbs	: MC_MoveAbsolute;
	_MCReset	: MC_Reset;
	_MCStop		: MC_Stop;
	_MCMoveVel	: MC_MoveVelocity;
	_MCPower	: MC_Power;
	_MCJog		: MC_Jog;
END_VAR

IF NOT __ISVALIDREF(Axis) THEN
	ErrorText := 'Axis Reference is Invalid.';
	RETURN;
ELSE
	ErrorText := '';
END_IF

_MCPower(Axis:= Axis,
			Enable:= TRUE,
			Enable_Positive:= TRUE,
			Enable_Negative:= TRUE,
			Override:= 100);
			
_MCReset(Axis:= Axis);
_MCStop(Axis:= Axis);
_MCMoveAbs(Axis:= Axis);
_MCMoveVel(Axis:= Axis);
_MCJog(Axis:= Axis);

Axis.ReadStatus();

METHOD M_Jog : BOOL
VAR_INPUT
	OwnerId : T_ResourceOwnerId;
	JogForward : BOOL;
	JogBackwards : BOOL;
	Mode : E_JogMode;
	Position : LREAL;
	Velocity : LREAL;
	Acceleration : LREAL;
	Deceleration : LREAL;
END_VAR

VAR_OUTPUT
	Done : BOOL;
	Error : BOOL;
	ErrorId : UDINT;
END_VAR
// Ignore commands from Services that do not own this BaseUnit.
M_Jog := FALSE;
Done := FALSE;
Error := FALSE;
ErrorId := 0;
IF NOT M_IsResourceOwner(OwnerId := OwnerId) THEN
	RETURN;
END_IF

_MCJog.JogForward := JogForward;
_MCJog.JogBackwards := JogBackwards;
_MCJog.Mode := Mode;
_MCJog.Position := Position;
_MCJog.Velocity := Velocity;
_MCJog.Acceleration := Acceleration;
_MCJog.Deceleration := Deceleration;

Done := _MCJog.Done;
Error := _MCJog.Error;
ErrorId := _MCJog.ErrorId;
M_Jog := TRUE;
END_METHOD

METHOD M_MoveAbs : BOOL
VAR_INPUT
	OwnerId : T_ResourceOwnerId;
	Execute : BOOL;
	Position : LREAL;
	Velocity : LREAL;
	Acceleration : LREAL;
	Deceleration : LREAL;
END_VAR

VAR_OUTPUT
	Done : BOOL;
	Error : BOOL;
END_VAR
// Ignore commands from Services that do not own this BaseUnit.
M_MoveAbs := FALSE;
Done := FALSE;
Error := FALSE;
IF NOT M_IsResourceOwner(OwnerId := OwnerId) THEN
	RETURN;
END_IF

_MCMoveAbs.Execute := Execute;
_MCMoveAbs.Position := Position;
_MCMoveAbs.Velocity := Velocity;
_MCMoveAbs.Acceleration := Acceleration;
_MCMoveAbs.Deceleration := Deceleration;

Done := _MCMoveAbs.Done;
Error := _MCMoveAbs.Error;
M_MoveAbs := TRUE;
END_METHOD

METHOD M_MoveVel : BOOL
VAR_INPUT
	OwnerId : T_ResourceOwnerId;
	Execute : BOOL;
	Param : ST_GCSpinAxisMoveVelParam;
END_VAR

VAR_OUTPUT
	InVelocity : BOOL;
	Error : BOOL;
END_VAR
// Ignore commands from Services that do not own this BaseUnit.
M_MoveVel := FALSE;
InVelocity := FALSE;
Error := FALSE;
IF NOT M_IsResourceOwner(OwnerId := OwnerId) THEN
	RETURN;
END_IF

_MCMoveVel.Execute := Execute;
IF Param.IsPositiveDirection THEN
	_MCMoveVel.Direction := MC_Direction.MC_Positive_Direction;
ELSE
	_MCMoveVel.Direction := MC_Direction.MC_Negative_Direction;
END_IF

_MCMoveVel.Velocity := Param.Velocity;
_MCMoveVel.Acceleration := Param.Acceleration;
_MCMoveVel.Deceleration := Param.Deceleration;

InVelocity := _MCMoveVel.InVelocity;
Error := _MCMoveVel.Error;
M_MoveVel := TRUE;
END_METHOD

METHOD M_Reset : BOOL
VAR_INPUT
	OwnerId : T_ResourceOwnerId;
	Execute : BOOL;
END_VAR

VAR_OUTPUT
	Done : BOOL;
	Error : BOOL;
END_VAR
// Ignore commands from Services that do not own this BaseUnit.
M_Reset := FALSE;
Done := FALSE;
Error := FALSE;
IF NOT M_IsResourceOwner(OwnerId := OwnerId) THEN
	RETURN;
END_IF

_MCReset.Execute := Execute;

Done := _MCReset.Done;
Error := _MCReset.Error;
M_Reset := TRUE;
END_METHOD

METHOD M_Stop : BOOL
VAR_INPUT
	OwnerId : T_ResourceOwnerId;
	Execute : BOOL;
	Deceleration : LREAL;
END_VAR

VAR_OUTPUT
	Done : BOOL;
	Error : BOOL;
END_VAR
// Ignore commands from Services that do not own this BaseUnit.
M_Stop := FALSE;
Done := FALSE;
Error := FALSE;
IF NOT M_IsResourceOwner(OwnerId := OwnerId) THEN
	RETURN;
END_IF

_MCStop.Execute := Execute;
_MCStop.Deceleration := Deceleration;

Done := _MCStop.Done;
Error := _MCStop.Error;
M_Stop := TRUE;
END_METHOD

PROPERTY PUBLIC AxisActualVelocity : LREAL
GET
// Expose motion feedback without exposing AXIS_REF to Services.
AxisActualVelocity := 0;
IF __ISVALIDREF(Axis) THEN
	AxisActualVelocity := Axis.NcToPlc.ActVelo;
END_IF
END_GET
END_PROPERTY

PROPERTY PUBLIC AxisHasJob : BOOL
GET
// Expose motion feedback without exposing AXIS_REF to Services.
AxisHasJob := FALSE;
IF __ISVALIDREF(Axis) THEN
	AxisHasJob := Axis.Status.HasJob;
END_IF
END_GET
END_PROPERTY

PROPERTY PUBLIC AxisIsDisabled : BOOL
GET
// Treat an invalid Axis reference as unavailable to callers.
AxisIsDisabled := TRUE;
IF __ISVALIDREF(Axis) THEN
	AxisIsDisabled := Axis.Status.Disabled;
END_IF
END_GET
END_PROPERTY

END_FUNCTION_BLOCK

// ---- POUs/00_BaseUnit/FB_BaseUnit.TcPOU
FUNCTION_BLOCK FB_BaseUnit
VAR
	// Owner ID zero means that no Service currently owns this BaseUnit.
	_ResourceOwnerId : T_ResourceOwnerId;
END_VAR

METHOD PUBLIC FINAL M_AcquireResource : BOOL
VAR_INPUT
	OwnerId : T_ResourceOwnerId;
END_VAR
// Reject zero because it represents the unowned state.
M_AcquireResource := FALSE;
IF OwnerId = 0 THEN
	RETURN;
END_IF

// Re-acquiring with the current Owner ID is intentionally idempotent.
IF (_ResourceOwnerId = 0) OR (_ResourceOwnerId = OwnerId) THEN
	_ResourceOwnerId := OwnerId;
	M_AcquireResource := TRUE;
END_IF
END_METHOD

METHOD PUBLIC FINAL M_IsResourceOwner : BOOL
VAR_INPUT
	OwnerId : T_ResourceOwnerId;
END_VAR
// Zero can never identify a valid Resource Owner.
M_IsResourceOwner := (OwnerId <> 0) AND (_ResourceOwnerId = OwnerId);
END_METHOD

METHOD PUBLIC FINAL M_ReleaseResource : BOOL
VAR_INPUT
	OwnerId : T_ResourceOwnerId;
END_VAR
// Only the current Owner may release the Resource.
M_ReleaseResource := FALSE;
IF NOT M_IsResourceOwner(OwnerId := OwnerId) THEN
	RETURN;
END_IF

_ResourceOwnerId := 0;
M_ReleaseResource := TRUE;
END_METHOD

PROPERTY PUBLIC FINAL ResourceIsAcquired : BOOL
GET
ResourceIsAcquired := _ResourceOwnerId <> 0;
END_GET
END_PROPERTY

PROPERTY PUBLIC FINAL ResourceOwnerId : T_ResourceOwnerId
GET
ResourceOwnerId := _ResourceOwnerId;
END_GET
END_PROPERTY

END_FUNCTION_BLOCK

// ---- POUs/10_Module/11_GC/Services/FB_GCSpinAxisJogServices.TcPOU
FUNCTION_BLOCK FB_GCSpinAxisJogServices EXTENDS FB_PackMLBase IMPLEMENTS I_ModuleServiceProperty
VAR_INPUT
	Ctrl : REFERENCE TO ST_GCSpinAxisJogCtrl;
	Status : REFERENCE TO ST_GCSpinAxisJogStatus;
	Axis_BaseUnit : REFERENCE TO FB_AxisControl;

	// The Module assigns a unique ID to this Service instance.
	ResourceOwnerId : T_ResourceOwnerId;
END_VAR

VAR_OUTPUT
END_VAR

VAR
	_StartOneShot	: R_TRIG;
	_ResetOneShot	: R_TRIG;
	_StopOneShot	: R_TRIG;
	_AbortOneShot	: R_TRIG;
	
	_ModuleMode		: T_PackMLMode;
END_VAR

// Update service state
Status.State := stOut.eStateCurrent;

A00_TrigCommand();

SUPER^();

ACTION A00_TrigCommand:
_StartOneShot(CLK:= Ctrl.Start);
IF _StartOneShot.Q THEN
	RequestCommand(E_PackMLCommand.Start);
END_IF

_ResetOneShot(CLK:= Ctrl.Reset);
IF _ResetOneShot.Q THEN
	RequestCommand(E_PackMLCommand.Reset);
END_IF

_StopOneShot(CLK:= Ctrl.Stop);
IF _StopOneShot.Q THEN
	RequestCommand(E_PackMLCommand.Stop);
END_IF

_AbortOneShot(CLK:= Ctrl.Abort);
IF _AbortOneShot.Q THEN
	RequestCommand(E_PackMLCommand.Abort);
END_IF
END_ACTION

METHOD PROTECTED H_OnAborted
VAR_INPUT
	bFirstScan	: BOOL;
END_VAR
// Release defensively in case an unexpected transition skipped cleanup.
Axis_BaseUnit.M_ReleaseResource(OwnerId := ResourceOwnerId);

Status.Busy := FALSE;
Status.Done := FALSE;
Status.Aborted := TRUE;

RequestCommand(E_PackMLCommand.Clear);
END_METHOD

METHOD PROTECTED H_OnAborting : E_PackMLHookResult
VAR_INPUT
	bFirstScan	: BOOL;
END_VAR
H_OnAborting := E_PackMLHookResult.Done;

// A Service that never acquired the Resource must not affect its Owner.
IF NOT Axis_BaseUnit.M_IsResourceOwner(OwnerId := ResourceOwnerId) THEN
	RETURN;
END_IF

Axis_BaseUnit.M_Jog(
	OwnerId:= ResourceOwnerId,
	JogForward:= FALSE, 
	JogBackwards:= FALSE, 
	Mode:= Ctrl.Param.Mode,
	Position:= Ctrl.Param.Position,
	Velocity:= Ctrl.Param.Velocity,
	Acceleration:= Ctrl.Param.Acceleration,
	Deceleration:= Ctrl.Param.Deceleration);

// Jog has no asynchronous abort phase once both direction commands are false.
Axis_BaseUnit.M_ReleaseResource(OwnerId := ResourceOwnerId);
END_METHOD

METHOD PROTECTED H_OnClearing : E_PackMLHookResult
VAR_INPUT
	bFirstScan	: BOOL;
END_VAR

VAR
	bServoOn : BOOL;
	bError : BOOL;
	nErrorId : UDINT;
END_VAR
H_OnClearing := E_PackMLHookResult.Done;
END_METHOD

METHOD PROTECTED H_OnComplete
VAR_INPUT
	bFirstScan	: BOOL;
END_VAR
// Completing normally releases first; this is an idempotent safety net.
Axis_BaseUnit.M_ReleaseResource(OwnerId := ResourceOwnerId);

Status.Busy := FALSE;
Status.Done := TRUE;
Status.Error := FALSE;
Status.Aborted := FALSE;
Status.ErrorId := E_GCSpinAxisJogErrorCode.None;

IF NOT Ctrl.Start THEN
	RequestCommand(E_PackMLCommand.Reset);
END_IF
END_METHOD

METHOD PROTECTED H_OnCompleting : E_PackMLHookResult
VAR_INPUT
	bFirstScan	: BOOL;
END_VAR
Status.Busy := FALSE;
Status.Done := TRUE;
Status.Error := FALSE;
Status.Aborted := FALSE;
Status.ErrorId := E_GCSpinAxisJogErrorCode.None;

Axis_BaseUnit.M_Jog(
	OwnerId:= ResourceOwnerId,
	JogForward:= FALSE, 
	JogBackwards:= FALSE, 
	Mode:= Ctrl.Param.Mode,
	Position:= Ctrl.Param.Position,
	Velocity:= Ctrl.Param.Velocity,
	Acceleration:= Ctrl.Param.Acceleration,
	Deceleration:= Ctrl.Param.Deceleration);

// Release only after the active Jog request has been withdrawn.
Axis_BaseUnit.M_ReleaseResource(OwnerId := ResourceOwnerId);
H_OnCompleting := E_PackMLHookResult.Done;
END_METHOD

METHOD PROTECTED H_OnExecute : E_PackMLHookResult
VAR_INPUT
	bFirstScan	: BOOL;
END_VAR

VAR
	bDone : BOOL;
	bError : BOOL;
END_VAR
H_OnExecute := E_PackMLHookResult.Busy;

Status.Busy := TRUE;
Status.Done := FALSE;
Status.Error := FALSE;
Status.Aborted := FALSE;
Status.ErrorId := E_GCSpinAxisJogErrorCode.None;

Axis_BaseUnit.M_Jog(
	OwnerId:= ResourceOwnerId,
	JogForward:= Ctrl.Param.JogForward,
	JogBackwards:= Ctrl.Param.JogBackwards,
	Mode:= Ctrl.Param.Mode,
	Position:= Ctrl.Param.Position,
	Velocity:= Ctrl.Param.Velocity,
	Acceleration:= Ctrl.Param.Acceleration,
	Deceleration:= Ctrl.Param.Deceleration,
	Done=> bDone, Error=> bError);


IF Ctrl.Param.Mode = E_JogMode.MC_JOGMODE_INCHING THEN
	IF bDone THEN
		Status.Busy := FALSE;
		Status.Done := TRUE;
		H_OnExecute := E_PackMLHookResult.Done;
		RETURN;
	END_IF
END_IF

IF bError THEN
		Status.Error := TRUE;
		Status.ErrorId := E_GCSpinAxisJogErrorCode.Jog_Error_During_Execute;
		
		RequestCommand(E_PackMLCommand.Stop);
END_IF
END_METHOD

METHOD PROTECTED H_OnHeld
VAR_INPUT
	bFirstScan	: BOOL;
END_VAR
// Default action hook intentionally empty. Override in derived FBs when needed.
END_METHOD

METHOD PROTECTED H_OnHolding : E_PackMLHookResult
VAR_INPUT
	bFirstScan	: BOOL;
END_VAR
// Default transient hooks complete immediately; override when work is required.
H_OnHolding := E_PackMLHookResult.Done;
END_METHOD

METHOD PROTECTED H_OnIdle
VAR_INPUT
	bFirstScan	: BOOL;
END_VAR
// Idle Services must not retain a Resource from an earlier operation.
Axis_BaseUnit.M_ReleaseResource(OwnerId := ResourceOwnerId);

Status.Busy := FALSE;
Status.Done := FALSE;
Status.Error := FALSE;
Status.Aborted := FALSE;
Status.ErrorId := E_GCSpinAxisJogErrorCode.None;
END_METHOD

METHOD PROTECTED H_OnResetting : E_PackMLHookResult
VAR_INPUT
	bFirstScan	: BOOL;
END_VAR
Status.Busy := FALSE;
Status.Done := FALSE;
Status.Error := FALSE;
Status.Aborted := FALSE;
Status.ErrorId := E_GCSpinAxisJogErrorCode.None;

H_OnResetting := E_PackMLHookResult.Done;
END_METHOD

METHOD PROTECTED H_OnStarting : E_PackMLHookResult
VAR_INPUT
	bFirstScan	: BOOL;
END_VAR
H_OnStarting := E_PackMLHookResult.Busy;

Status.Busy := TRUE;
Status.Done := FALSE;
Status.Error := FALSE;
Status.Aborted := FALSE;
Status.ErrorId := E_GCSpinAxisJogErrorCode.None;

// Validate Service-owned data before reserving the shared BaseUnit.
IF (Ctrl.Param.JogBackwards AND Ctrl.Param.JogForward) OR
	(NOT Ctrl.Param.JogBackwards AND NOT Ctrl.Param.JogForward) OR
	Ctrl.Param.Velocity = 0 THEN
	Status.Error:= TRUE;
	Status.ErrorId:= E_GCSpinAxisJogErrorCode.Invalid_Param;
	RequestCommand(E_PackMLCommand.Stop);
	RETURN;
END_IF

// Resource contention is a failed Start, not a wait condition.
IF NOT Axis_BaseUnit.M_AcquireResource(OwnerId := ResourceOwnerId) THEN
	Status.Error := TRUE;
	Status.ErrorId := E_GCSpinAxisJogErrorCode.Resource_Acquire_Failed_During_Starting;
	RequestCommand(E_PackMLCommand.Stop);
	RETURN;
END_IF

// Physical checks occur only after this Service owns the BaseUnit.
IF Axis_BaseUnit.AxisIsDisabled THEN
	Status.Error:= TRUE;
	Status.ErrorId:= E_GCSpinAxisJogErrorCode.Axis_Not_Servo_On_During_Starting;
	RequestCommand(E_PackMLCommand.Abort);
	RETURN;
END_IF

IF Axis_BaseUnit.AxisHasJob THEN
	Status.Error:= TRUE;
	Status.ErrorId:= E_GCSpinAxisJogErrorCode.Axis_Is_Busy_During_Starting;
	RequestCommand(E_PackMLCommand.Stop);
	RETURN;
END_IF

H_OnStarting := E_PackMLHookResult.Done;
END_METHOD

METHOD PROTECTED H_OnStopped
VAR_INPUT
	bFirstScan	: BOOL;
END_VAR
// Release defensively after every Stop path.
Axis_BaseUnit.M_ReleaseResource(OwnerId := ResourceOwnerId);

Status.Busy := FALSE;
Status.Done := FALSE;
Status.Aborted := TRUE;
END_METHOD

METHOD PROTECTED H_OnStopping : E_PackMLHookResult
VAR_INPUT
	bFirstScan	: BOOL;
END_VAR
H_OnStopping := E_PackMLHookResult.Done;

// Resource acquisition failures enter Stopping without owning the Axis.
IF NOT Axis_BaseUnit.M_IsResourceOwner(OwnerId := ResourceOwnerId) THEN
	RETURN;
END_IF

Axis_BaseUnit.M_Jog(
	OwnerId:= ResourceOwnerId,
	JogForward:= FALSE, 
	JogBackwards:= FALSE, 
	Mode:= Ctrl.Param.Mode,
	Position:= Ctrl.Param.Position,
	Velocity:= Ctrl.Param.Velocity,
	Acceleration:= Ctrl.Param.Acceleration,
	Deceleration:= Ctrl.Param.Deceleration);

// Jog is stopped once both direction commands have been withdrawn.
Axis_BaseUnit.M_ReleaseResource(OwnerId := ResourceOwnerId);
END_METHOD

METHOD PROTECTED H_OnSuspended
VAR_INPUT
	bFirstScan	: BOOL;
END_VAR
// Default action hook intentionally empty. Override in derived FBs when needed.
END_METHOD

METHOD PROTECTED H_OnSuspending : E_PackMLHookResult
VAR_INPUT
	bFirstScan	: BOOL;
END_VAR
// Default transient hooks complete immediately; override when work is required.
H_OnSuspending := E_PackMLHookResult.Done;
END_METHOD

METHOD PROTECTED H_OnUndefined : E_PackMLHookResult
VAR_INPUT
	bFirstScan	: BOOL;
END_VAR
// The base FB leaves Undefined immediately unless a derived FB delays startup.
H_OnUndefined := E_PackMLHookResult.Done;
END_METHOD

METHOD PROTECTED H_OnUnholding : E_PackMLHookResult
VAR_INPUT
	bFirstScan	: BOOL;
END_VAR
// Default transient hooks complete immediately; override when work is required.
H_OnUnholding := E_PackMLHookResult.Done;
END_METHOD

METHOD PROTECTED H_OnUnsuspending : E_PackMLHookResult
VAR_INPUT
	bFirstScan	: BOOL;
END_VAR
// Default transient hooks complete immediately; override when work is required.
H_OnUnsuspending := E_PackMLHookResult.Done;
END_METHOD

PROPERTY ModuleMode : T_PackMLMode
GET
ModuleMode := _ModuleMode;
END_GET
SET
_ModuleMode := ModuleMode;
END_SET
END_PROPERTY

END_FUNCTION_BLOCK

// ---- POUs/10_Module/11_GC/Services/FB_GCSpinAxisMoveAbsServices.TcPOU
FUNCTION_BLOCK FB_GCSpinAxisMoveAbsServices EXTENDS FB_PackMLBase IMPLEMENTS I_ModuleServiceProperty
VAR_INPUT
	Ctrl : REFERENCE TO ST_GCSpinAxisMoveAbsCtrl;
	Status : REFERENCE TO ST_GCSpinAxisMoveAbsStatus;
	Axis_BaseUnit : REFERENCE TO FB_AxisControl;
	// The Module assigns a unique ID to this Service instance.
	ResourceOwnerId : T_ResourceOwnerId;
END_VAR

VAR_OUTPUT
END_VAR

VAR
	_StartOneShot	: R_TRIG;
	_ResetOneShot	: R_TRIG;
	_StopOneShot	: R_TRIG;
	_AbortOneShot	: R_TRIG;
	
	_ModuleMode		: T_PackMLMode;
END_VAR

// Update service state
Status.State := stOut.eStateCurrent;

A00_TrigCommand();

SUPER^();

ACTION A00_TrigCommand:
_StartOneShot(CLK:= Ctrl.Start);
IF _StartOneShot.Q THEN
	RequestCommand(E_PackMLCommand.Start);
END_IF

_ResetOneShot(CLK:= Ctrl.Reset);
IF _ResetOneShot.Q THEN
	RequestCommand(E_PackMLCommand.Reset);
END_IF

_StopOneShot(CLK:= Ctrl.Stop);
IF _StopOneShot.Q THEN
	RequestCommand(E_PackMLCommand.Stop);
END_IF

_AbortOneShot(CLK:= Ctrl.Abort);
IF _AbortOneShot.Q THEN
	RequestCommand(E_PackMLCommand.Abort);
END_IF
END_ACTION

METHOD PROTECTED H_OnAborted
VAR_INPUT
	bFirstScan	: BOOL;
END_VAR
// Release defensively in case an unexpected transition skipped cleanup.
Axis_BaseUnit.M_ReleaseResource(OwnerId := ResourceOwnerId);

Status.Busy := FALSE;
Status.Done := FALSE;
Status.Aborted := TRUE;

RequestCommand(E_PackMLCommand.Clear);
END_METHOD

METHOD PROTECTED H_OnAborting : E_PackMLHookResult
VAR_INPUT
	bFirstScan	: BOOL;
END_VAR

VAR
	bDone : BOOL;
	bError : BOOL;
END_VAR
H_OnAborting := E_PackMLHookResult.Busy;

// A Service that never acquired the Resource must not reset its Owner's Axis.
IF NOT Axis_BaseUnit.M_IsResourceOwner(OwnerId := ResourceOwnerId) THEN
	H_OnAborting := E_PackMLHookResult.Done;
	RETURN;
END_IF

// Withdraw MoveAbsolute before resetting the Axis.
Axis_BaseUnit.M_MoveAbs(
	OwnerId := ResourceOwnerId,
	Execute := FALSE,
	Position:= Ctrl.Param.Position,
	Velocity:= Ctrl.Param.Velocity,
	Acceleration:= Ctrl.Param.Acceleration,
	Deceleration:= Ctrl.Param.Deceleration);
	
Axis_BaseUnit.M_Reset(
	OwnerId := ResourceOwnerId,
	Execute := TRUE,
	Done=> bDone, Error=> bError);

IF bDone THEN
	Axis_BaseUnit.M_Reset(
		OwnerId := ResourceOwnerId,
		Execute := FALSE);
	// Keep ownership until the asynchronous Reset has completed.
	Axis_BaseUnit.M_ReleaseResource(OwnerId := ResourceOwnerId);
	H_OnAborting := E_PackMLHookResult.Done;
END_IF
END_METHOD

METHOD PROTECTED H_OnClearing : E_PackMLHookResult
VAR_INPUT
	bFirstScan	: BOOL;
END_VAR

VAR
	bServoOn : BOOL;
	bError : BOOL;
	nErrorId : UDINT;
END_VAR
H_OnClearing := E_PackMLHookResult.Done;
END_METHOD

METHOD PROTECTED H_OnComplete
VAR_INPUT
	bFirstScan	: BOOL;
END_VAR
// Completing normally releases first; this is an idempotent safety net.
Axis_BaseUnit.M_ReleaseResource(OwnerId := ResourceOwnerId);

Status.Busy := FALSE;
Status.Done := TRUE;
Status.Error := FALSE;
Status.Aborted := FALSE;
Status.ErrorId := E_GCSpinAxisMoveAbsErrorCode.None;

IF NOT Ctrl.Start THEN
	RequestCommand(E_PackMLCommand.Reset);
END_IF
END_METHOD

METHOD PROTECTED H_OnCompleting : E_PackMLHookResult
VAR_INPUT
	bFirstScan	: BOOL;
END_VAR
Status.Busy := FALSE;
Status.Done := TRUE;
Status.Error := FALSE;
Status.Aborted := FALSE;
Status.ErrorId := E_GCSpinAxisMoveAbsErrorCode.None;

Axis_BaseUnit.M_MoveAbs(
	OwnerId:= ResourceOwnerId,
	Execute:= FALSE,
	Position:= Ctrl.Param.Position,
	Velocity:= Ctrl.Param.Velocity,
	Acceleration:= Ctrl.Param.Acceleration,
	Deceleration:= Ctrl.Param.Deceleration);

// Release only after the active MoveAbsolute request has been withdrawn.
Axis_BaseUnit.M_ReleaseResource(OwnerId := ResourceOwnerId);
H_OnCompleting := E_PackMLHookResult.Done;
END_METHOD

METHOD PROTECTED H_OnExecute : E_PackMLHookResult
VAR_INPUT
	bFirstScan	: BOOL;
END_VAR

VAR
	bDone : BOOL;
	bError : BOOL;
END_VAR
H_OnExecute := E_PackMLHookResult.Busy;

Status.Busy := TRUE;
Status.Done := FALSE;
Status.Error := FALSE;
Status.Aborted := FALSE;
Status.ErrorId := E_GCSpinAxisMoveAbsErrorCode.None;

Axis_BaseUnit.M_MoveAbs(
	OwnerId:= ResourceOwnerId,
	Execute:= TRUE,
	Position:= Ctrl.Param.Position,
	Velocity:= Ctrl.Param.Velocity,
	Acceleration:= Ctrl.Param.Acceleration,
	Deceleration:= Ctrl.Param.Deceleration,
	Done=> bDone, Error=> bError);


IF bDone THEN
	Status.Busy := FALSE;
	Status.Done := TRUE;
	H_OnExecute := E_PackMLHookResult.Done;
	RETURN;
END_IF

IF bError THEN
		Status.Error := TRUE;
		Status.ErrorId := E_GCSpinAxisMoveAbsErrorCode.MoveAbs_Error_During_Execute;
		
		RequestCommand(E_PackMLCommand.Stop);
END_IF
END_METHOD

METHOD PROTECTED H_OnHeld
VAR_INPUT
	bFirstScan	: BOOL;
END_VAR
// Default action hook intentionally empty. Override in derived FBs when needed.
END_METHOD

METHOD PROTECTED H_OnHolding : E_PackMLHookResult
VAR_INPUT
	bFirstScan	: BOOL;
END_VAR
// Default transient hooks complete immediately; override when work is required.
H_OnHolding := E_PackMLHookResult.Done;
END_METHOD

METHOD PROTECTED H_OnIdle
VAR_INPUT
	bFirstScan	: BOOL;
END_VAR
// Idle Services must not retain a Resource from an earlier operation.
Axis_BaseUnit.M_ReleaseResource(OwnerId := ResourceOwnerId);

Status.Busy := FALSE;
Status.Done := FALSE;
Status.Error := FALSE;
Status.Aborted := FALSE;
Status.ErrorId := E_GCSpinAxisMoveAbsErrorCode.None;
END_METHOD

METHOD PROTECTED H_OnResetting : E_PackMLHookResult
VAR_INPUT
	bFirstScan	: BOOL;
END_VAR
Status.Busy := FALSE;
Status.Done := FALSE;
Status.Error := FALSE;
Status.Aborted := FALSE;
Status.ErrorId := E_GCSpinAxisMoveAbsErrorCode.None;

H_OnResetting := E_PackMLHookResult.Done;
END_METHOD

METHOD PROTECTED H_OnStarting : E_PackMLHookResult
VAR_INPUT
	bFirstScan	: BOOL;
END_VAR
H_OnStarting := E_PackMLHookResult.Busy;

Status.Busy := TRUE;
Status.Done := FALSE;
Status.Error := FALSE;
Status.Aborted := FALSE;
Status.ErrorId := E_GCSpinAxisMoveAbsErrorCode.None;

// Validate Service-owned data before reserving the shared BaseUnit.
IF Ctrl.Param.Velocity <= 0 THEN
	Status.Error:= TRUE;
	Status.ErrorId:= E_GCSpinAxisMoveAbsErrorCode.Invalid_Param;
	RequestCommand(E_PackMLCommand.Stop);
	RETURN;
END_IF

// Resource contention is a failed Start, not a wait condition.
IF NOT Axis_BaseUnit.M_AcquireResource(OwnerId := ResourceOwnerId) THEN
	Status.Error := TRUE;
	Status.ErrorId := E_GCSpinAxisMoveAbsErrorCode.Resource_Acquire_Failed_During_Starting;
	RequestCommand(E_PackMLCommand.Stop);
	RETURN;
END_IF

// Physical checks occur only after this Service owns the BaseUnit.
IF Axis_BaseUnit.AxisIsDisabled THEN
	Status.Error:= TRUE;
	Status.ErrorId:= E_GCSpinAxisMoveAbsErrorCode.Axis_Not_Servo_On_During_Starting;
	RequestCommand(E_PackMLCommand.Abort);
	RETURN;
END_IF

IF Axis_BaseUnit.AxisHasJob THEN
	Status.Error:= TRUE;
	Status.ErrorId:= E_GCSpinAxisMoveAbsErrorCode.Axis_Is_Busy_During_Starting;
	RequestCommand(E_PackMLCommand.Stop);
	RETURN;
END_IF

H_OnStarting := E_PackMLHookResult.Done;
END_METHOD

METHOD PROTECTED H_OnStopped
VAR_INPUT
	bFirstScan	: BOOL;
END_VAR
// Release defensively after every Stop path.
Axis_BaseUnit.M_ReleaseResource(OwnerId := ResourceOwnerId);

Status.Busy := FALSE;
Status.Done := FALSE;
Status.Aborted := TRUE;
END_METHOD

METHOD PROTECTED H_OnStopping : E_PackMLHookResult
VAR_INPUT
	bFirstScan	: BOOL;
END_VAR

VAR
	bDone : BOOL;
	bError : BOOL;
END_VAR
H_OnStopping := E_PackMLHookResult.Busy;

// Resource acquisition failures enter Stopping without owning the Axis.
IF NOT Axis_BaseUnit.M_IsResourceOwner(OwnerId := ResourceOwnerId) THEN
	H_OnStopping := E_PackMLHookResult.Done;
	RETURN;
END_IF

// Withdraw MoveAbsolute before issuing the physical Stop.
Axis_BaseUnit.M_MoveAbs(
	OwnerId := ResourceOwnerId,
	Execute := FALSE,
	Position:= Ctrl.Param.Position,
	Velocity:= Ctrl.Param.Velocity,
	Acceleration:= Ctrl.Param.Acceleration,
	Deceleration:= Ctrl.Param.Deceleration);
	
Axis_BaseUnit.M_Stop(
	OwnerId := ResourceOwnerId,
	Execute := TRUE, 
	Deceleration:= Ctrl.Param.Deceleration,
	Done=> bDone, Error=> bError);

IF bDone THEN
	Axis_BaseUnit.M_Stop(
		OwnerId := ResourceOwnerId,
		Execute := FALSE, 
		Deceleration:= Ctrl.Param.Deceleration);
	// Ownership is released only after the asynchronous Stop has completed.
	Axis_BaseUnit.M_ReleaseResource(OwnerId := ResourceOwnerId);
	H_OnStopping := E_PackMLHookResult.Done;
	
ELSIF bError THEN
	// Throw up error
	Status.Error := TRUE;
	Status.ErrorId := E_GCSpinAxisMoveAbsErrorCode.Error_While_Stop_Axis;
	
	Axis_BaseUnit.M_Stop(
		OwnerId := ResourceOwnerId,
		Execute := FALSE, 
		Deceleration:= Ctrl.Param.Deceleration);
		
	RequestCommand(E_PackMLCommand.Abort);
END_IF
END_METHOD

METHOD PROTECTED H_OnSuspended
VAR_INPUT
	bFirstScan	: BOOL;
END_VAR
// Default action hook intentionally empty. Override in derived FBs when needed.
END_METHOD

METHOD PROTECTED H_OnSuspending : E_PackMLHookResult
VAR_INPUT
	bFirstScan	: BOOL;
END_VAR
// Default transient hooks complete immediately; override when work is required.
H_OnSuspending := E_PackMLHookResult.Done;
END_METHOD

METHOD PROTECTED H_OnUndefined : E_PackMLHookResult
VAR_INPUT
	bFirstScan	: BOOL;
END_VAR
// The base FB leaves Undefined immediately unless a derived FB delays startup.
H_OnUndefined := E_PackMLHookResult.Done;
END_METHOD

METHOD PROTECTED H_OnUnholding : E_PackMLHookResult
VAR_INPUT
	bFirstScan	: BOOL;
END_VAR
// Default transient hooks complete immediately; override when work is required.
H_OnUnholding := E_PackMLHookResult.Done;
END_METHOD

METHOD PROTECTED H_OnUnsuspending : E_PackMLHookResult
VAR_INPUT
	bFirstScan	: BOOL;
END_VAR
// Default transient hooks complete immediately; override when work is required.
H_OnUnsuspending := E_PackMLHookResult.Done;
END_METHOD

PROPERTY ModuleMode : T_PackMLMode
GET
ModuleMode := _ModuleMode;
END_GET
SET
_ModuleMode := ModuleMode;
END_SET
END_PROPERTY

END_FUNCTION_BLOCK

// ---- POUs/10_Module/11_GC/Services/FB_GCSpinAxisMoveVelServices.TcPOU
FUNCTION_BLOCK FB_GCSpinAxisMoveVelServices EXTENDS FB_PackMLBase IMPLEMENTS I_ModuleServiceProperty
VAR_INPUT
	Ctrl : REFERENCE TO ST_GCSpinAxisMoveVelCtrl;
	Status : REFERENCE TO ST_GCSpinAxisMoveVelStatus;
	Axis_BaseUnit : REFERENCE TO FB_AxisControl;
	// The Module assigns a unique ID to this Service instance.
	ResourceOwnerId : T_ResourceOwnerId;
END_VAR

VAR_OUTPUT
END_VAR

VAR
	_StartOneShot	: R_TRIG;
	_ResetOneShot	: R_TRIG;
	_StopOneShot	: R_TRIG;
	_AbortOneShot	: R_TRIG;
	
	_ModuleMode		: T_PackMLMode;
END_VAR

// Update service state
Status.State := stOut.eStateCurrent;
Status.ActVel := Axis_BaseUnit.AxisActualVelocity;
A00_TrigCommand();

SUPER^();

ACTION A00_TrigCommand:
_StartOneShot(CLK:= Ctrl.Start);
IF _StartOneShot.Q THEN
	RequestCommand(E_PackMLCommand.Start);
END_IF

_ResetOneShot(CLK:= Ctrl.Reset);
IF _ResetOneShot.Q THEN
	RequestCommand(E_PackMLCommand.Reset);
END_IF

_StopOneShot(CLK:= Ctrl.Stop);
IF _StopOneShot.Q THEN
	RequestCommand(E_PackMLCommand.Stop);
END_IF

_AbortOneShot(CLK:= Ctrl.Abort);
IF _AbortOneShot.Q THEN
	RequestCommand(E_PackMLCommand.Abort);
END_IF
END_ACTION

METHOD PROTECTED H_OnAborted
VAR_INPUT
	bFirstScan	: BOOL;
END_VAR
// Release defensively in case an unexpected transition skipped cleanup.
Axis_BaseUnit.M_ReleaseResource(OwnerId := ResourceOwnerId);

Status.Busy := FALSE;
Status.Done := FALSE;
Status.Aborted := TRUE;

RequestCommand(E_PackMLCommand.Clear);
END_METHOD

METHOD PROTECTED H_OnAborting : E_PackMLHookResult
VAR_INPUT
	bFirstScan	: BOOL;
END_VAR

VAR
	bDone : BOOL;
	bError : BOOL;
END_VAR
H_OnAborting := E_PackMLHookResult.Busy;

// A Service that never acquired the Resource must not reset its Owner's Axis.
IF NOT Axis_BaseUnit.M_IsResourceOwner(OwnerId := ResourceOwnerId) THEN
	H_OnAborting := E_PackMLHookResult.Done;
	RETURN;
END_IF

// Withdraw MoveVelocity before resetting the Axis.
Axis_BaseUnit.M_MoveVel(
	OwnerId := ResourceOwnerId,
	Execute := FALSE,
	Ctrl.Param);
	
Axis_BaseUnit.M_Reset(
	OwnerId := ResourceOwnerId,
	Execute := TRUE,
	Done=> bDone, Error=> bError);

IF bDone THEN
	Axis_BaseUnit.M_Reset(
		OwnerId := ResourceOwnerId,
		Execute := FALSE);
	// Keep ownership until the asynchronous Reset has completed.
	Axis_BaseUnit.M_ReleaseResource(OwnerId := ResourceOwnerId);
	H_OnAborting := E_PackMLHookResult.Done;
END_IF
END_METHOD

METHOD PROTECTED H_OnClearing : E_PackMLHookResult
VAR_INPUT
	bFirstScan	: BOOL;
END_VAR

VAR
	bServoOn : BOOL;
	bError : BOOL;
	nErrorId : UDINT;
END_VAR
H_OnClearing := E_PackMLHookResult.Done;
END_METHOD

METHOD PROTECTED H_OnComplete
VAR_INPUT
	bFirstScan	: BOOL;
END_VAR
// Completing normally releases first; this is an idempotent safety net.
Axis_BaseUnit.M_ReleaseResource(OwnerId := ResourceOwnerId);

Status.Busy := FALSE;
Status.Done := TRUE;
Status.Error := FALSE;
Status.Aborted := FALSE;
Status.ErrorId := E_GCSpinAxisMoveVelErrorCode.None;

IF NOT Ctrl.Start THEN
	RequestCommand(E_PackMLCommand.Reset);
END_IF
END_METHOD

METHOD PROTECTED H_OnCompleting : E_PackMLHookResult
VAR_INPUT
	bFirstScan	: BOOL;
END_VAR
Status.Busy := FALSE;
Status.Done := TRUE;
Status.Error := FALSE;
Status.Aborted := FALSE;
Status.ErrorId := E_GCSpinAxisMoveVelErrorCode.None;

Axis_BaseUnit.M_MoveVel(
	OwnerId:= ResourceOwnerId,
	Execute:= FALSE,
	Param := Ctrl.Param);

// Release only after the active MoveVelocity request has been withdrawn.
Axis_BaseUnit.M_ReleaseResource(OwnerId := ResourceOwnerId);
H_OnCompleting := E_PackMLHookResult.Done;
END_METHOD

METHOD PROTECTED H_OnExecute : E_PackMLHookResult
VAR_INPUT
	bFirstScan	: BOOL;
END_VAR

VAR
	bDone : BOOL;
	bError : BOOL;
END_VAR
H_OnExecute := E_PackMLHookResult.Busy;

Status.Busy := TRUE;
Status.Done := FALSE;
Status.Error := FALSE;
Status.Aborted := FALSE;
Status.ErrorId := E_GCSpinAxisMoveVelErrorCode.None;

Axis_BaseUnit.M_MoveVel(
	OwnerId:= ResourceOwnerId,
	Execute:= TRUE,
	Param:= Ctrl.Param,
	InVelocity=> bDone, Error=> bError);


IF bDone THEN
	Status.Busy := FALSE;
	Status.Done := TRUE;
	H_OnExecute := E_PackMLHookResult.Done;
	RETURN;
END_IF

IF bError THEN
		Status.Error := TRUE;
		Status.ErrorId := E_GCSpinAxisMoveVelErrorCode.MoveVel_Error_During_Execute;
		
		RequestCommand(E_PackMLCommand.Stop);
END_IF
END_METHOD

METHOD PROTECTED H_OnHeld
VAR_INPUT
	bFirstScan	: BOOL;
END_VAR
// Default action hook intentionally empty. Override in derived FBs when needed.
END_METHOD

METHOD PROTECTED H_OnHolding : E_PackMLHookResult
VAR_INPUT
	bFirstScan	: BOOL;
END_VAR
// Default transient hooks complete immediately; override when work is required.
H_OnHolding := E_PackMLHookResult.Done;
END_METHOD

METHOD PROTECTED H_OnIdle
VAR_INPUT
	bFirstScan	: BOOL;
END_VAR
// Idle Services must not retain a Resource from an earlier operation.
Axis_BaseUnit.M_ReleaseResource(OwnerId := ResourceOwnerId);

Status.Busy := FALSE;
Status.Done := FALSE;
Status.Error := FALSE;
Status.Aborted := FALSE;
Status.ErrorId := E_GCSpinAxisMoveVelErrorCode.None;
END_METHOD

METHOD PROTECTED H_OnResetting : E_PackMLHookResult
VAR_INPUT
	bFirstScan	: BOOL;
END_VAR
Status.Busy := FALSE;
Status.Done := FALSE;
Status.Error := FALSE;
Status.Aborted := FALSE;
Status.ErrorId := E_GCSpinAxisMoveVelErrorCode.None;

H_OnResetting := E_PackMLHookResult.Done;
END_METHOD

METHOD PROTECTED H_OnStarting : E_PackMLHookResult
VAR_INPUT
	bFirstScan	: BOOL;
END_VAR
H_OnStarting := E_PackMLHookResult.Busy;

Status.Busy := TRUE;
Status.Done := FALSE;
Status.Error := FALSE;
Status.Aborted := FALSE;
Status.ErrorId := E_GCSpinAxisMoveVelErrorCode.None;

// Validate Service-owned data before reserving the shared BaseUnit.
IF Ctrl.Param.Velocity <= 0 THEN
	Status.Error:= TRUE;
	Status.ErrorId:= E_GCSpinAxisMoveVelErrorCode.Invalid_Param;
	RequestCommand(E_PackMLCommand.Stop);
	RETURN;
END_IF

// Resource contention is a failed Start, not a wait condition.
IF NOT Axis_BaseUnit.M_AcquireResource(OwnerId := ResourceOwnerId) THEN
	Status.Error := TRUE;
	Status.ErrorId := E_GCSpinAxisMoveVelErrorCode.Resource_Acquire_Failed_During_Starting;
	RequestCommand(E_PackMLCommand.Stop);
	RETURN;
END_IF

// Physical checks occur only after this Service owns the BaseUnit.
IF Axis_BaseUnit.AxisIsDisabled THEN
	Status.Error:= TRUE;
	Status.ErrorId:= E_GCSpinAxisMoveVelErrorCode.Axis_Not_Servo_On_During_Starting;
	RequestCommand(E_PackMLCommand.Abort);
	RETURN;
END_IF

IF Axis_BaseUnit.AxisHasJob THEN
	Status.Error:= TRUE;
	Status.ErrorId:= E_GCSpinAxisMoveVelErrorCode.Axis_Is_Busy_During_Starting;
	RequestCommand(E_PackMLCommand.Stop);
	RETURN;
END_IF

H_OnStarting := E_PackMLHookResult.Done;
END_METHOD

METHOD PROTECTED H_OnStopped
VAR_INPUT
	bFirstScan	: BOOL;
END_VAR
// Release defensively after every Stop path.
Axis_BaseUnit.M_ReleaseResource(OwnerId := ResourceOwnerId);

Status.Busy := FALSE;
Status.Done := FALSE;
Status.Aborted := TRUE;
END_METHOD

METHOD PROTECTED H_OnStopping : E_PackMLHookResult
VAR_INPUT
	bFirstScan	: BOOL;
END_VAR

VAR
	bDone : BOOL;
	bError : BOOL;
END_VAR
H_OnStopping := E_PackMLHookResult.Busy;

// Resource acquisition failures enter Stopping without owning the Axis.
IF NOT Axis_BaseUnit.M_IsResourceOwner(OwnerId := ResourceOwnerId) THEN
	H_OnStopping := E_PackMLHookResult.Done;
	RETURN;
END_IF

// Withdraw MoveVelocity before issuing the physical Stop.
Axis_BaseUnit.M_MoveVel(
	OwnerId := ResourceOwnerId,
	Execute := FALSE,
	Param:= Ctrl.Param);
	
Axis_BaseUnit.M_Stop(
	OwnerId := ResourceOwnerId,
	Execute := TRUE, 
	Deceleration:= Ctrl.Param.Deceleration,
	Done=> bDone, Error=> bError);

IF bDone THEN
	Axis_BaseUnit.M_Stop(
		OwnerId := ResourceOwnerId,
		Execute := FALSE, 
		Deceleration:= Ctrl.Param.Deceleration);
	// Ownership is released only after the asynchronous Stop has completed.
	Axis_BaseUnit.M_ReleaseResource(OwnerId := ResourceOwnerId);
	H_OnStopping := E_PackMLHookResult.Done;
	
ELSIF bError THEN
	// Throw up error
	Status.Error := TRUE;
	Status.ErrorId := E_GCSpinAxisMoveVelErrorCode.Error_While_Stop_Axis;
	
	Axis_BaseUnit.M_Stop(
		OwnerId := ResourceOwnerId,
		Execute := FALSE, 
		Deceleration:= Ctrl.Param.Deceleration);
		
	RequestCommand(E_PackMLCommand.Abort);
END_IF
END_METHOD

METHOD PROTECTED H_OnSuspended
VAR_INPUT
	bFirstScan	: BOOL;
END_VAR
// Default action hook intentionally empty. Override in derived FBs when needed.
END_METHOD

METHOD PROTECTED H_OnSuspending : E_PackMLHookResult
VAR_INPUT
	bFirstScan	: BOOL;
END_VAR
// Default transient hooks complete immediately; override when work is required.
H_OnSuspending := E_PackMLHookResult.Done;
END_METHOD

METHOD PROTECTED H_OnUndefined : E_PackMLHookResult
VAR_INPUT
	bFirstScan	: BOOL;
END_VAR
// The base FB leaves Undefined immediately unless a derived FB delays startup.
H_OnUndefined := E_PackMLHookResult.Done;
END_METHOD

METHOD PROTECTED H_OnUnholding : E_PackMLHookResult
VAR_INPUT
	bFirstScan	: BOOL;
END_VAR
// Default transient hooks complete immediately; override when work is required.
H_OnUnholding := E_PackMLHookResult.Done;
END_METHOD

METHOD PROTECTED H_OnUnsuspending : E_PackMLHookResult
VAR_INPUT
	bFirstScan	: BOOL;
END_VAR
// Default transient hooks complete immediately; override when work is required.
H_OnUnsuspending := E_PackMLHookResult.Done;
END_METHOD

PROPERTY ModuleMode : T_PackMLMode
GET
ModuleMode := _ModuleMode;
END_GET
SET
_ModuleMode := ModuleMode;
END_SET
END_PROPERTY

END_FUNCTION_BLOCK
